LIN {X 0,Y 456.186,Z 1038.193,A -85,B 0,C 180,E1 14833.103,E2 14833.103} C_VEL
LIN {X 0,Y 454.706,Z 1048.98,A -85,B 0,C 180,E1 14838.466,E2 14838.466} C_VEL
LIN {X 0,Y 454.201,Z 1053.772,A -85,B 0,C 180,E1 14842.332,E2 14842.332} C_VEL
LIN {X 0,Y 454.081,Z 1056.363,A -85,B 0,C 180,E1 14848.088,E2 14848.088} C_VEL
LIN {X 0,Y 454.216,Z 1055.013,A -85,B 0,C 180,E1 14851.913,E2 14851.913} C_VEL
LIN {X 0,Y 454.611,Z 1049.888,A -85,B 0,C 180,E1 14856.701,E2 14856.701} C_VEL
LIN {X 0,Y 456.014,Z 1038.504,A -85,B 0,C 180,E1 14862.475,E2 14862.475} C_VEL
LIN {X 0,Y 459.25,Z 1020.736,A -85,B 0,C 180,E1 14868.27,E2 14868.27} C_VEL
LIN {X 0,Y 464.709,Z 997.367,A -85,B 0,C 180,E1 14873.669,E2 14873.669} C_VEL
LIN {X 0,Y 471.743,Z 970.349,A -85,B 0,C 180,E1 14878.315,E2 14878.315} C_VEL
LIN {X 0,Y 480.458,Z 937.273,A -85,B 0,C 180,E1 14882.614,E2 14882.614} C_VEL
LIN {X 0,Y 489.598,Z 900.461,A -85,B 0,C 180,E1 14886.199,E2 14886.199} C_VEL
LIN {X 0,Y 498.715,Z 857.606,A -85,B 0,C 180,E1 14889.265,E2 14889.265} C_VEL
LIN {X 0,Y 506.278,Z 812.153,A -85,B 0,C 180,E1 14891.552,E2 14891.552} C_VEL
LIN {X 0,Y 492.603,Z 777.017,A -85,B 0,C 180,E1 14894.833,E2 14894.833} C_VEL
LIN {X 0,Y 474.285,Z 742.388,A -85,B 0,C 180,E1 14898.475,E2 14898.475} C_VEL
LIN {X 0,Y 454.825,Z 713.013,A -85,B 0,C 180,E1 14902.271,E2 14902.271} C_VEL
LIN {X 0,Y 452.383,Z 707.31,A -85,B 0,C 180,E1 14902.914,E2 14902.914} C_VEL
LIN {X 0,Y 452.524,Z 707.31,A -85,B 0,C 180,E1 14909.843,E2 14909.843} C_VEL
LIN {X 0,Y 452.661,Z 707.31,A -85,B 0,C 180,E1 14916.31,E2 14916.31} C_VEL
LIN {X 0,Y 452.928,Z 707.31,A -85,B 0,C 180,E1 14922.472,E2 14922.472} C_VEL
LIN {X 0,Y 453.411,Z 707.31,A -85,B 0,C 180,E1 14928.428,E2 14928.428} C_VEL
LIN {X 0,Y 453.726,Z 707.31,A -85,B 0,C 180,E1 14934.246,E2 14934.246} C_VEL
LIN {X 0,Y 453.754,Z 707.31,A -85,B 0,C 180,E1 14941.91,E2 14941.91} C_VEL
LIN {X 0,Y 453.568,Z 707.31,A -85,B 0,C 180,E1 14947.677,E2 14947.677} C_VEL
LIN {X 0,Y 453.098,Z 707.31,A -85,B 0,C 180,E1 14954.087,E2 14954.087} C_VEL
LIN {X 0,Y 452.724,Z 707.31,A -85,B 0,C 180,E1 14960.404,E2 14960.404} C_VEL
LIN {X 0,Y 452.601,Z 707.31,A -85,B 0,C 180,E1 14965.798,E2 14965.798} C_VEL
LIN {X 0,Y 452.45,Z 707.31,A -85,B 0,C 180,E1 14972.4,E2 14972.4} C_VEL
LIN {X 0,Y 452.465,Z 708.154,A -85,B 0,C 180,E1 14974.776,E2 14974.776} C_VEL
LIN {X 0,Y 455.588,Z 713.626,A -85,B 0,C 180,E1 14975.457,E2 14975.457} C_VEL
LIN {X 0,Y 478.519,Z 749.077,A -85,B 0,C 180,E1 14979.815,E2 14979.815} C_VEL
LIN {X 0,Y 497.384,Z 784.719,A -85,B 0,C 180,E1 14983.272,E2 14983.272} C_VEL
LIN {X 0,Y 508.29,Z 812.813,A -85,B 0,C 180,E1 14985.653,E2 14985.653} C_VEL
LIN {X 0,Y 501.832,Z 855.362,A -85,B 0,C 180,E1 14987.392,E2 14987.392} C_VEL
LIN {X 0,Y 493.956,Z 895.887,A -85,B 0,C 180,E1 14989.745,E2 14989.745} C_VEL
LIN {X 0,Y 484.639,Z 936.283,A -85,B 0,C 180,E1 14992.968,E2 14992.968} C_VEL
LIN {X 0,Y 475.031,Z 974.706,A -85,B 0,C 180,E1 14997.157,E2 14997.157} C_VEL
LIN {X 0,Y 466.793,Z 1007.142,A -85,B 0,C 180,E1 15001.917,E2 15001.917} C_VEL
LIN {X 0,Y 460.332,Z 1035.051,A -85,B 0,C 180,E1 15007.471,E2 15007.471} C_VEL
LIN {X 0,Y 456.522,Z 1055.517,A -85,B 0,C 180,E1 15013.115,E2 15013.115} C_VEL
LIN {X 0,Y 454.835,Z 1068.915,A -85,B 0,C 180,E1 15018.468,E2 15018.468} C_VEL
LIN {X 0,Y 454.297,Z 1076.636,A -85,B 0,C 180,E1 15023.295,E2 15023.295} C_VEL
LIN {X 0,Y 454.154,Z 1080.28,A -85,B 0,C 180,E1 15028.087,E2 15028.087} C_VEL
LIN {X 0,Y 454.299,Z 1080.303,A -85,B 0,C 180,E1 15031.911,E2 15031.911} C_VEL
LIN {X 0,Y 454.27,Z 1075.566,A -85,B 0,C 180,E1 15037.667,E2 15037.667} C_VEL
LIN {X 0,Y 454.36,Z 1074.281,A -85,B 0,C 180,E1 15038.648,E2 15038.648} C_VEL
LIN {X 0,Y 450.707,Z 1070.833,A -85,B 0,C 180,E1 15040.771,E2 15040.771} C_VEL
LIN {X 0,Y 447.241,Z 1066.661,A -85,B 0,C 180,E1 15042.912,E2 15042.912} C_VEL
LIN {X 0,Y 449.59,Z 1051.412,A -85,B 0,C 180,E1 15048.62,E2 15048.62} C_VEL
LIN {X 0,Y 454.024,Z 1030.563,A -85,B 0,C 180,E1 15054.133,E2 15054.133} C_VEL
LIN {X 0,Y 460.882,Z 1004.236,A -85,B 0,C 180,E1 15059.28,E2 15059.28} C_VEL
LIN {X 0,Y 470.006,Z 971.713,A -85,B 0,C 180,E1 15064.022,E2 15064.022} C_VEL
LIN {X 0,Y 479.765,Z 935.941,A -85,B 0,C 180,E1 15067.932,E2 15067.932} C_VEL
LIN {X 0,Y 489.925,Z 894.816,A -85,B 0,C 180,E1 15071.239,E2 15071.239} C_VEL
LIN {X 0,Y 499.025,Z 850.387,A -85,B 0,C 180,E1 15073.79,E2 15073.79} C_VEL
LIN {X 0,Y 504.38,Z 814.102,A -85,B 0,C 180,E1 15075.308,E2 15075.308} C_VEL
LIN {X 0,Y 489.342,Z 779.423,A -85,B 0,C 180,E1 15078.711,E2 15078.711} C_VEL
LIN {X 0,Y 469.19,Z 744.618,A -85,B 0,C 180,E1 15082.806,E2 15082.806} C_VEL
LIN {X 0,Y 451.64,Z 719.415,A -85,B 0,C 180,E1 15086.659,E2 15086.659} C_VEL
LIN {X 0,Y 447.451,Z 713.438,A -85,B 0,C 180,E1 15087.687,E2 15087.687} C_VEL
LIN {X 0,Y 444.607,Z 708.574,A -85,B 0,C 180,E1 15088.439,E2 15088.439} C_VEL
LIN {X 0,Y 444.514,Z 707.31,A -85,B 0,C 180,E1 15088.637,E2 15088.637} C_VEL
LIN {X 0,Y 444.625,Z 707.31,A -85,B 0,C 180,E1 15093.704,E2 15093.704} C_VEL
LIN {X 0,Y 444.826,Z 707.31,A -85,B 0,C 180,E1 15100.086,E2 15100.086} C_VEL
LIN {X 0,Y 445.231,Z 707.31,A -85,B 0,C 180,E1 15106.22,E2 15106.22} C_VEL
LIN {X 0,Y 445.633,Z 707.31,A -85,B 0,C 180,E1 15112.186,E2 15112.186} C_VEL
LIN {X 0,Y 445.832,Z 707.31,A -85,B 0,C 180,E1 15118.056,E2 15118.056} C_VEL
LIN {X 0,Y 445.563,Z 707.31,A -85,B 0,C 180,E1 15123.904,E2 15123.904} C_VEL
LIN {X 0,Y 445.331,Z 707.31,A -85,B 0,C 180,E1 15129.8,E2 15129.8} C_VEL
LIN {X 0,Y 445.045,Z 707.31,A -85,B 0,C 180,E1 15135.811,E2 15135.811} C_VEL
LIN {X 0,Y 444.85,Z 707.31,A -85,B 0,C 180,E1 15142.01,E2 15142.01} C_VEL
LIN {X 0,Y 444.556,Z 707.31,A -85,B 0,C 180,E1 15149.224,E2 15149.224} C_VEL
LIN {X 0,Y 444.568,Z 707.532,A -85,B 0,C 180,E1 15149.854,E2 15149.854} C_VEL
LIN {X 0,Y 446.931,Z 712.981,A -85,B 0,C 180,E1 15150.524,E2 15150.524} C_VEL
LIN {X 0,Y 449.765,Z 716.523,A -85,B 0,C 180,E1 15151.214,E2 15151.214} C_VEL
LIN {X 0,Y 467.8,Z 742.864,A -85,B 0,C 180,E1 15155.295,E2 15155.295} C_VEL
LIN {X 0,Y 485.366,Z 773.688,A -85,B 0,C 180,E1 15159.154,E2 15159.154} C_VEL
LIN {X 0,Y 500.292,Z 808.905,A -85,B 0,C 180,E1 15162.897,E2 15162.897} C_VEL
LIN {X 0,Y 502.326,Z 818.223,A -85,B 0,C 180,E1 15163.698,E2 15163.698} C_VEL
LIN {X 0,Y 494.118,Z 861.819,A -85,B 0,C 180,E1 15165.968,E2 15165.968} C_VEL
LIN {X 0,Y 484.618,Z 902.54,A -85,B 0,C 180,E1 15168.955,E2 15168.955} C_VEL
LIN {X 0,Y 474.394,Z 940.654,A -85,B 0,C 180,E1 15172.785,E2 15172.785} C_VEL
LIN {X 0,Y 464.358,Z 975.438,A -85,B 0,C 180,E1 15177.533,E2 15177.533} C_VEL
LIN {X 0,Y 456.413,Z 1003.839,A -85,B 0,C 180,E1 15182.821,E2 15182.821} C_VEL
LIN {X 0,Y 450.631,Z 1027.018,A -85,B 0,C 180,E1 15188.808,E2 15188.808} C_VEL
LIN {X 0,Y 447.82,Z 1042.419,A -85,B 0,C 180,E1 15194.587,E2 15194.587} C_VEL
LIN {X 0,Y 446.526,Z 1051.875,A -85,B 0,C 180,E1 15200.231,E2 15200.231} C_VEL
LIN {X 0,Y 446.125,Z 1056.308,A -85,B 0,C 180,E1 15206.105,E2 15206.105} C_VEL
LIN {X 0,Y 446.415,Z 1056.23,A -85,B 0,C 180,E1 15210.001,E2 15210.001} C_VEL
LIN {X 0,Y 446.59,Z 1051.43,A -85,B 0,C 180,E1 15215.844,E2 15215.844} C_VEL
LIN {X 0,Y 447.898,Z 1041.018,A -85,B 0,C 180,E1 15221.713,E2 15221.713} C_VEL
LIN {X 0,Y 450.99,Z 1024.433,A -85,B 0,C 180,E1 15227.604,E2 15227.604} C_VEL
LIN {X 0,Y 456.366,Z 1001.802,A -85,B 0,C 180,E1 15233.224,E2 15233.224} C_VEL
LIN {X 0,Y 463.843,Z 973.876,A -85,B 0,C 180,E1 15238.306,E2 15238.306} C_VEL
LIN {X 0,Y 473.106,Z 940.161,A -85,B 0,C 180,E1 15242.856,E2 15242.856} C_VEL
LIN {X 0,Y 483.21,Z 900.916,A -85,B 0,C 180,E1 15246.756,E2 15246.756} C_VEL
LIN {X 0,Y 492.663,Z 857.898,A -85,B 0,C 180,E1 15249.862,E2 15249.862} C_VEL
LIN {X 0,Y 500.04,Z 814.852,A -85,B 0,C 180,E1 15252.07,E2 15252.07} C_VEL
LIN {X 0,Y 486.137,Z 778.648,A -85,B 0,C 180,E1 15255.57,E2 15255.57} C_VEL
LIN {X 0,Y 467.182,Z 743.055,A -85,B 0,C 180,E1 15259.499,E2 15259.499} C_VEL
LIN {X 0,Y 447.132,Z 713.195,A -85,B 0,C 180,E1 15263.624,E2 15263.624} C_VEL
LIN {X 0,Y 444.506,Z 708.118,A -85,B 0,C 180,E1 15264.25,E2 15264.25} C_VEL
LIN {X 0,Y 444.531,Z 707.31,A -85,B 0,C 180,E1 15269.243,E2 15269.243} C_VEL
LIN {X 0,Y 444.743,Z 707.31,A -85,B 0,C 180,E1 15275.862,E2 15275.862} C_VEL
LIN {X 0,Y 445.023,Z 707.31,A -85,B 0,C 180,E1 15282.454,E2 15282.454} C_VEL
LIN {X 0,Y 445.484,Z 707.31,A -85,B 0,C 180,E1 15288.22,E2 15288.22} C_VEL
LIN {X 0,Y 445.805,Z 707.31,A -85,B 0,C 180,E1 15294.143,E2 15294.143} C_VEL
LIN {X 0,Y 445.841,Z 707.31,A -85,B 0,C 180,E1 15301.944,E2 15301.944} C_VEL
LIN {X 0,Y 445.647,Z 707.31,A -85,B 0,C 180,E1 15307.814,E2 15307.814} C_VEL
LIN {X 0,Y 445.244,Z 707.31,A -85,B 0,C 180,E1 15313.779,E2 15313.779} C_VEL
LIN {X 0,Y 444.836,Z 707.31,A -85,B 0,C 180,E1 15319.913,E2 15319.913} C_VEL
LIN {X 0,Y 444.632,Z 707.31,A -85,B 0,C 180,E1 15326.295,E2 15326.295} C_VEL
LIN {X 0,Y 444.507,Z 707.31,A -85,B 0,C 180,E1 15333.284,E2 15333.284} C_VEL
LIN {X 0,Y 446.827,Z 712.942,A -85,B 0,C 180,E1 15333.896,E2 15333.896} C_VEL
LIN {X 0,Y 449.926,Z 717.277,A -85,B 0,C 180,E1 15334.572,E2 15334.572} C_VEL
LIN {X 0,Y 468.229,Z 744.574,A -85,B 0,C 180,E1 15338.234,E2 15338.234} C_VEL
LIN {X 0,Y 488.407,Z 781.004,A -85,B 0,C 180,E1 15342.056,E2 15342.056} C_VEL
LIN {X 0,Y 502.202,Z 814.372,A -85,B 0,C 180,E1 15345.071,E2 15345.071} C_VEL
LIN {X 0,Y 495.094,Z 859.617,A -85,B 0,C 180,E1 15346.999,E2 15346.999} C_VEL
LIN {X 0,Y 487.037,Z 898.739,A -85,B 0,C 180,E1 15349.362,E2 15349.362} C_VEL
LIN {X 0,Y 477.602,Z 938.053,A -85,B 0,C 180,E1 15352.589,E2 15352.589} C_VEL
LIN {X 0,Y 468.18,Z 974.379,A -85,B 0,C 180,E1 15356.615,E2 15356.615} C_VEL
LIN {X 0,Y 459.534,Z 1006.996,A -85,B 0,C 180,E1 15361.463,E2 15361.463} C_VEL
LIN {X 0,Y 453.069,Z 1033.593,A -85,B 0,C 180,E1 15366.801,E2 15366.801} C_VEL
LIN {X 0,Y 448.77,Z 1055.256,A -85,B 0,C 180,E1 15372.813,E2 15372.813} C_VEL
LIN {X 0,Y 446.971,Z 1068.675,A -85,B 0,C 180,E1 15378.262,E2 15378.262} C_VEL
LIN {X 0,Y 446.409,Z 1076.408,A -85,B 0,C 180,E1 15383.176,E2 15383.176} C_VEL
LIN {X 0,Y 446.252,Z 1080.066,A -85,B 0,C 180,E1 15388.053,E2 15388.053} C_VEL
LIN {X 0,Y 446.395,Z 1080.094,A -85,B 0,C 180,E1 15391.945,E2 15391.945} C_VEL
LIN {X 0,Y 446.375,Z 1075.37,A -85,B 0,C 180,E1 15397.804,E2 15397.804} C_VEL
LIN {X 0,Y 447.241,Z 1066.661,A -85,B 0,C 180,E1 15402.912,E2 15402.912} C_VEL
LIN {X 0,Y 443.939,Z 1061.938,A -85,B 0,C 180,E1 15405.041,E2 15405.041} C_VEL
LIN {X 0,Y 440.957,Z 1056.558,A -85,B 0,C 180,E1 15407.179,E2 15407.179} C_VEL
LIN {X 0,Y 445.138,Z 1036.482,A -85,B 0,C 180,E1 15413.104,E2 15413.104} C_VEL
LIN {X 0,Y 451.671,Z 1011.412,A -85,B 0,C 180,E1 15418.479,E2 15418.479} C_VEL
LIN {X 0,Y 460.159,Z 982.234,A -85,B 0,C 180,E1 15423.166,E2 15423.166} C_VEL
LIN {X 0,Y 470.066,Z 947.885,A -85,B 0,C 180,E1 15427.334,E2 15427.334} C_VEL
LIN {X 0,Y 480.939,Z 906.832,A -85,B 0,C 180,E1 15431.004,E2 15431.004} C_VEL
LIN {X 0,Y 490.884,Z 863.211,A -85,B 0,C 180,E1 15433.786,E2 15433.786} C_VEL
LIN {X 0,Y 498.525,Z 817.345,A -85,B 0,C 180,E1 15435.837,E2 15435.837} C_VEL
LIN {X 0,Y 483.899,Z 783.034,A -85,B 0,C 180,E1 15439.334,E2 15439.334} C_VEL
LIN {X 0,Y 465.253,Z 750.222,A -85,B 0,C 180,E1 15443.315,E2 15443.315} C_VEL
LIN {X 0,Y 444.926,Z 720.523,A -85,B 0,C 180,E1 15448.004,E2 15448.004} C_VEL
LIN {X 0,Y 439.645,Z 713.508,A -85,B 0,C 180,E1 15449.383,E2 15449.383} C_VEL
LIN {X 0,Y 436.726,Z 708.582,A -85,B 0,C 180,E1 15450.22,E2 15450.22} C_VEL
LIN {X 0,Y 436.609,Z 707.31,A -85,B 0,C 180,E1 15450.436,E2 15450.436} C_VEL
LIN {X 0,Y 436.827,Z 707.31,A -85,B 0,C 180,E1 15457.571,E2 15457.571} C_VEL
LIN {X 0,Y 437.121,Z 707.31,A -85,B 0,C 180,E1 15463.902,E2 15463.902} C_VEL
LIN {X 0,Y 437.639,Z 707.31,A -85,B 0,C 180,E1 15470.034,E2 15470.034} C_VEL
LIN {X 0,Y 437.672,Z 707.31,A -85,B 0,C 180,E1 15476.033,E2 15476.033} C_VEL
LIN {X 0,Y 437.618,Z 707.31,A -85,B 0,C 180,E1 15481.988,E2 15481.988} C_VEL
LIN {X 0,Y 437.455,Z 707.31,A -85,B 0,C 180,E1 15487.968,E2 15487.968} C_VEL
LIN {X 0,Y 437.277,Z 707.31,A -85,B 0,C 180,E1 15494.043,E2 15494.043} C_VEL
LIN {X 0,Y 436.933,Z 707.31,A -85,B 0,C 180,E1 15500.542,E2 15500.542} C_VEL
LIN {X 0,Y 436.643,Z 707.31,A -85,B 0,C 180,E1 15507.476,E2 15507.476} C_VEL
LIN {X 0,Y 436.677,Z 708.191,A -85,B 0,C 180,E1 15508.089,E2 15508.089} C_VEL
LIN {X 0,Y 439.613,Z 713.446,A -85,B 0,C 180,E1 15508.942,E2 15508.942} C_VEL
LIN {X 0,Y 442.067,Z 716.673,A -85,B 0,C 180,E1 15509.593,E2 15509.593} C_VEL
LIN {X 0,Y 459.278,Z 741.265,A -85,B 0,C 180,E1 15513.764,E2 15513.764} C_VEL
LIN {X 0,Y 477.735,Z 772.896,A -85,B 0,C 180,E1 15518.011,E2 15518.011} C_VEL
LIN {X 0,Y 492.517,Z 807.026,A -85,B 0,C 180,E1 15521.828,E2 15521.828} C_VEL
LIN {X 0,Y 496.591,Z 819.004,A -85,B 0,C 180,E1 15523.066,E2 15523.066} C_VEL
LIN {X 0,Y 488.32,Z 861.92,A -85,B 0,C 180,E1 15525.323,E2 15525.323} C_VEL
LIN {X 0,Y 478.532,Z 902.526,A -85,B 0,C 180,E1 15528.317,E2 15528.317} C_VEL
LIN {X 0,Y 467.903,Z 940.684,A -85,B 0,C 180,E1 15532.179,E2 15532.179} C_VEL
LIN {X 0,Y 457.703,Z 974.903,A -85,B 0,C 180,E1 15536.888,E2 15536.888} C_VEL
LIN {X 0,Y 449.079,Z 1004.023,A -85,B 0,C 180,E1 15542.356,E2 15542.356} C_VEL
LIN {X 0,Y 443.037,Z 1027.164,A -85,B 0,C 180,E1 15548.427,E2 15548.427} C_VEL
LIN {X 0,Y 440.099,Z 1041.922,A -85,B 0,C 180,E1 15554.011,E2 15554.011} C_VEL
LIN {X 0,Y 438.821,Z 1050.866,A -85,B 0,C 180,E1 15559.052,E2 15559.052} C_VEL
LIN {X 0,Y 438.263,Z 1055.639,A -85,B 0,C 180,E1 15564.047,E2 15564.047} C_VEL
LIN {X 0,Y 438.533,Z 1056.446,A -85,B 0,C 180,E1 15570.001,E2 15570.001} C_VEL
LIN {X 0,Y 438.724,Z 1051.669,A -85,B 0,C 180,E1 15575.949,E2 15575.949} C_VEL
LIN {X 0,Y 439.819,Z 1043.03,A -85,B 0,C 180,E1 15581.15,E2 15581.15} C_VEL
LIN {X 0,Y 443.037,Z 1026.246,A -85,B 0,C 180,E1 15587.471,E2 15587.471} C_VEL
LIN {X 0,Y 448.683,Z 1003.307,A -85,B 0,C 180,E1 15593.382,E2 15593.382} C_VEL
LIN {X 0,Y 456.726,Z 974.533,A -85,B 0,C 180,E1 15598.736,E2 15598.736} C_VEL
LIN {X 0,Y 466.408,Z 940.559,A -85,B 0,C 180,E1 15603.389,E2 15603.389} C_VEL
LIN {X 0,Y 476.835,Z 901.541,A -85,B 0,C 180,E1 15607.312,E2 15607.312} C_VEL
LIN {X 0,Y 486.484,Z 859.193,A -85,B 0,C 180,E1 15610.413,E2 15610.413} C_VEL
LIN {X 0,Y 493.876,Z 817.882,A -85,B 0,C 180,E1 15612.569,E2 15612.569} C_VEL
LIN {X 0,Y 480.27,Z 781.639,A -85,B 0,C 180,E1 15616.201,E2 15616.201} C_VEL
LIN {X 0,Y 462.388,Z 747.702,A -85,B 0,C 180,E1 15620.099,E2 15620.099} C_VEL
LIN {X 0,Y 443.563,Z 719.344,A -85,B 0,C 180,E1 15624.113,E2 15624.113} C_VEL
LIN {X 0,Y 439,Z 713.014,A -85,B 0,C 180,E1 15625.17,E2 15625.17} C_VEL
LIN {X 0,Y 436.537,Z 707.31,A -85,B 0,C 180,E1 15626.008,E2 15626.008} C_VEL
LIN {X 0,Y 436.697,Z 707.31,A -85,B 0,C 180,E1 15633.181,E2 15633.181} C_VEL
LIN {X 0,Y 436.905,Z 707.31,A -85,B 0,C 180,E1 15639.702,E2 15639.702} C_VEL
LIN {X 0,Y 437.383,Z 707.31,A -85,B 0,C 180,E1 15645.961,E2 15645.961} C_VEL
LIN {X 0,Y 437.749,Z 707.31,A -85,B 0,C 180,E1 15652.037,E2 15652.037} C_VEL
LIN {X 0,Y 437.643,Z 707.31,A -85,B 0,C 180,E1 15658.012,E2 15658.012} C_VEL
LIN {X 0,Y 437.67,Z 707.31,A -85,B 0,C 180,E1 15663.967,E2 15663.967} C_VEL
LIN {X 0,Y 437.653,Z 707.31,A -85,B 0,C 180,E1 15669.966,E2 15669.966} C_VEL
LIN {X 0,Y 437.133,Z 707.31,A -85,B 0,C 180,E1 15676.097,E2 15676.097} C_VEL
LIN {X 0,Y 436.839,Z 707.31,A -85,B 0,C 180,E1 15682.428,E2 15682.428} C_VEL
LIN {X 0,Y 436.644,Z 707.31,A -85,B 0,C 180,E1 15689.066,E2 15689.066} C_VEL
LIN {X 0,Y 436.634,Z 707.318,A -85,B 0,C 180,E1 15691.773,E2 15691.773} C_VEL
LIN {X 0,Y 438.701,Z 712.684,A -85,B 0,C 180,E1 15692.344,E2 15692.344} C_VEL
LIN {X 0,Y 441.686,Z 716.541,A -85,B 0,C 180,E1 15693.035,E2 15693.035} C_VEL
LIN {X 0,Y 461.26,Z 745.525,A -85,B 0,C 180,E1 15697.188,E2 15697.188} C_VEL
LIN {X 0,Y 480.502,Z 779.804,A -85,B 0,C 180,E1 15701.003,E2 15701.003} C_VEL
LIN {X 0,Y 495.946,Z 816.725,A -85,B 0,C 180,E1 15704.492,E2 15704.492} C_VEL
LIN {X 0,Y 488.248,Z 864.434,A -85,B 0,C 180,E1 15706.629,E2 15706.629} C_VEL
LIN {X 0,Y 478.889,Z 907.156,A -85,B 0,C 180,E1 15709.373,E2 15709.373} C_VEL
LIN {X 0,Y 468.621,Z 947.439,A -85,B 0,C 180,E1 15712.965,E2 15712.965} C_VEL
LIN {X 0,Y 458.67,Z 983.652,A -85,B 0,C 180,E1 15717.358,E2 15717.358} C_VEL
LIN {X 0,Y 450.507,Z 1013.662,A -85,B 0,C 180,E1 15722.251,E2 15722.251} C_VEL
LIN {X 0,Y 444.354,Z 1038.417,A -85,B 0,C 180,E1 15727.66,E2 15727.66} C_VEL
LIN {X 0,Y 440.773,Z 1056.435,A -85,B 0,C 180,E1 15733.007,E2 15733.007} C_VEL
LIN {X 0,Y 438.995,Z 1069.765,A -85,B 0,C 180,E1 15738.729,E2 15738.729} C_VEL
LIN {X 0,Y 438.483,Z 1077.216,A -85,B 0,C 180,E1 15744.048,E2 15744.048} C_VEL
LIN {X 0,Y 438.512,Z 1080.206,A -85,B 0,C 180,E1 15749.999,E2 15749.999} C_VEL
LIN {X 0,Y 438.47,Z 1077.374,A -85,B 0,C 180,E1 15755.95,E2 15755.95} C_VEL
LIN {X 0,Y 438.943,Z 1070.23,A -85,B 0,C 180,E1 15761.235,E2 15761.235} C_VEL
LIN {X 0,Y 440.957,Z 1056.558,A -85,B 0,C 180,E1 15767.179,E2 15767.179} C_VEL
LIN {X 0,Y 438.256,Z 1050.682,A -85,B 0,C 180,E1 15769.303,E2 15769.303} C_VEL
LIN {X 0,Y 435.819,Z 1044.111,A -85,B 0,C 180,E1 15771.419,E2 15771.419} C_VEL
LIN {X 0,Y 441.902,Z 1020.734,A -85,B 0,C 180,E1 15777.102,E2 15777.102} C_VEL
LIN {X 0,Y 449.922,Z 993.481,A -85,B 0,C 180,E1 15782.037,E2 15782.037} C_VEL
LIN {X 0,Y 460.181,Z 959.48,A -85,B 0,C 180,E1 15786.645,E2 15786.645} C_VEL
LIN {X 0,Y 471.284,Z 920.476,A -85,B 0,C 180,E1 15790.54,E2 15790.54} C_VEL
LIN {X 0,Y 482.028,Z 877.609,A -85,B 0,C 180,E1 15793.621,E2 15793.621} C_VEL
LIN {X 0,Y 491.151,Z 832.43,A -85,B 0,C 180,E1 15795.87,E2 15795.87} C_VEL
LIN {X 0,Y 492.497,Z 819.986,A -85,B 0,C 180,E1 15796.421,E2 15796.421} C_VEL
LIN {X 0,Y 478.235,Z 786.157,A -85,B 0,C 180,E1 15800.004,E2 15800.004} C_VEL
LIN {X 0,Y 460.352,Z 754.369,A -85,B 0,C 180,E1 15804.033,E2 15804.033} C_VEL
LIN {X 0,Y 441.618,Z 726.789,A -85,B 0,C 180,E1 15808.523,E2 15808.523} C_VEL
LIN {X 0,Y 432.417,Z 713.971,A -85,B 0,C 180,E1 15811.08,E2 15811.08} C_VEL
LIN {X 0,Y 428.934,Z 709.282,A -85,B 0,C 180,E1 15812.131,E2 15812.131} C_VEL
LIN {X 0,Y 428.702,Z 707.31,A -85,B 0,C 180,E1 15812.414,E2 15812.414} C_VEL
LIN {X 0,Y 428.939,Z 707.31,A -85,B 0,C 180,E1 15819.316,E2 15819.316} C_VEL
LIN {X 0,Y 429.337,Z 707.31,A -85,B 0,C 180,E1 15825.7,E2 15825.7} C_VEL
LIN {X 0,Y 429.79,Z 707.31,A -85,B 0,C 180,E1 15831.896,E2 15831.896} C_VEL
LIN {X 0,Y 430.011,Z 707.31,A -85,B 0,C 180,E1 15837.984,E2 15837.984} C_VEL
LIN {X 0,Y 429.74,Z 707.31,A -85,B 0,C 180,E1 15844.048,E2 15844.048} C_VEL
LIN {X 0,Y 429.498,Z 707.31,A -85,B 0,C 180,E1 15850.165,E2 15850.165} C_VEL
LIN {X 0,Y 429.163,Z 707.31,A -85,B 0,C 180,E1 15856.412,E2 15856.412} C_VEL
LIN {X 0,Y 428.901,Z 707.31,A -85,B 0,C 180,E1 15863.275,E2 15863.275} C_VEL
LIN {X 0,Y 428.772,Z 707.433,A -85,B 0,C 180,E1 15866.094,E2 15866.094} C_VEL
LIN {X 0,Y 430.827,Z 712.624,A -85,B 0,C 180,E1 15866.808,E2 15866.808} C_VEL
LIN {X 0,Y 434.1,Z 716.27,A -85,B 0,C 180,E1 15867.744,E2 15867.744} C_VEL
LIN {X 0,Y 451.862,Z 741.347,A -85,B 0,C 180,E1 15872.382,E2 15872.382} C_VEL
LIN {X 0,Y 470.793,Z 773.323,A -85,B 0,C 180,E1 15876.968,E2 15876.968} C_VEL
LIN {X 0,Y 485.624,Z 807.281,A -85,B 0,C 180,E1 15880.947,E2 15880.947} C_VEL
LIN {X 0,Y 490.548,Z 822.804,A -85,B 0,C 180,E1 15882.573,E2 15882.573} C_VEL
LIN {X 0,Y 482.12,Z 863.975,A -85,B 0,C 180,E1 15884.79,E2 15884.79} C_VEL
LIN {X 0,Y 472.154,Z 903.798,A -85,B 0,C 180,E1 15887.78,E2 15887.78} C_VEL
LIN {X 0,Y 461.125,Z 941.939,A -85,B 0,C 180,E1 15891.703,E2 15891.703} C_VEL
LIN {X 0,Y 450.846,Z 974.977,A -85,B 0,C 180,E1 15896.318,E2 15896.318} C_VEL
LIN {X 0,Y 441.817,Z 1004.137,A -85,B 0,C 180,E1 15901.862,E2 15901.862} C_VEL
LIN {X 0,Y 435.485,Z 1027.311,A -85,B 0,C 180,E1 15908.034,E2 15908.034} C_VEL
LIN {X 0,Y 432.126,Z 1043.636,A -85,B 0,C 180,E1 15914.427,E2 15914.427} C_VEL
LIN {X 0,Y 430.784,Z 1052.48,A -85,B 0,C 180,E1 15920.073,E2 15920.073} C_VEL
LIN {X 0,Y 430.342,Z 1056.723,A -85,B 0,C 180,E1 15925.962,E2 15925.962} C_VEL
LIN {X 0,Y 430.632,Z 1056.661,A -85,B 0,C 180,E1 15930.001,E2 15930.001} C_VEL
LIN {X 0,Y 430.843,Z 1051.908,A -85,B 0,C 180,E1 15936.058,E2 15936.058} C_VEL
LIN {X 0,Y 431.986,Z 1043.515,A -85,B 0,C 180,E1 15941.254,E2 15941.254} C_VEL
LIN {X 0,Y 435.344,Z 1026.723,A -85,B 0,C 180,E1 15947.734,E2 15947.734} C_VEL
LIN {X 0,Y 441.287,Z 1003.631,A -85,B 0,C 180,E1 15953.798,E2 15953.798} C_VEL
LIN {X 0,Y 449.747,Z 974.698,A -85,B 0,C 180,E1 15959.259,E2 15959.259} C_VEL
LIN {X 0,Y 459.731,Z 940.957,A -85,B 0,C 180,E1 15963.94,E2 15963.94} C_VEL
LIN {X 0,Y 470.543,Z 901.992,A -85,B 0,C 180,E1 15967.898,E2 15967.898} C_VEL
LIN {X 0,Y 480.557,Z 859.406,A -85,B 0,C 180,E1 15971.043,E2 15971.043} C_VEL
LIN {X 0,Y 487.619,Z 820.313,A -85,B 0,C 180,E1 15973.135,E2 15973.135} C_VEL
LIN {X 0,Y 474.166,Z 784.229,A -85,B 0,C 180,E1 15976.888,E2 15976.888} C_VEL
LIN {X 0,Y 456.53,Z 750.238,A -85,B 0,C 180,E1 15980.954,E2 15980.954} C_VEL
LIN {X 0,Y 436.596,Z 720.251,A -85,B 0,C 180,E1 15985.435,E2 15985.435} C_VEL
LIN {X 0,Y 431.409,Z 713.289,A -85,B 0,C 180,E1 15986.714,E2 15986.714} C_VEL
LIN {X 0,Y 428.731,Z 708.643,A -85,B 0,C 180,E1 15987.438,E2 15987.438} C_VEL
LIN {X 0,Y 428.644,Z 707.31,A -85,B 0,C 180,E1 15987.701,E2 15987.701} C_VEL
LIN {X 0,Y 428.835,Z 707.31,A -85,B 0,C 180,E1 15994.906,E2 15994.906} C_VEL
LIN {X 0,Y 429.087,Z 707.31,A -85,B 0,C 180,E1 16001.463,E2 16001.463} C_VEL
LIN {X 0,Y 429.601,Z 707.31,A -85,B 0,C 180,E1 16007.777,E2 16007.777} C_VEL
LIN {X 0,Y 429.96,Z 707.31,A -85,B 0,C 180,E1 16013.927,E2 16013.927} C_VEL
LIN {X 0,Y 430.02,Z 707.31,A -85,B 0,C 180,E1 16022.016,E2 16022.016} C_VEL
LIN {X 0,Y 429.72,Z 707.31,A -85,B 0,C 180,E1 16029.095,E2 16029.095} C_VEL
LIN {X 0,Y 429.35,Z 707.31,A -85,B 0,C 180,E1 16034.3,E2 16034.3} C_VEL
LIN {X 0,Y 428.95,Z 707.31,A -85,B 0,C 180,E1 16040.684,E2 16040.684} C_VEL
LIN {X 0,Y 428.7,Z 707.31,A -85,B 0,C 180,E1 16047.904,E2 16047.904} C_VEL
LIN {X 0,Y 428.744,Z 708.006,A -85,B 0,C 180,E1 16050.127,E2 16050.127} C_VEL
LIN {X 0,Y 431.498,Z 713.334,A -85,B 0,C 180,E1 16050.889,E2 16050.889} C_VEL
LIN {X 0,Y 434.188,Z 717.076,A -85,B 0,C 180,E1 16051.565,E2 16051.565} C_VEL
LIN {X 0,Y 452.302,Z 743.403,A -85,B 0,C 180,E1 16055.673,E2 16055.673} C_VEL
LIN {X 0,Y 471.39,Z 776.156,A -85,B 0,C 180,E1 16059.636,E2 16059.636} C_VEL
LIN {X 0,Y 486.953,Z 811.593,A -85,B 0,C 180,E1 16063.202,E2 16063.202} C_VEL
LIN {X 0,Y 489.952,Z 820.648,A -85,B 0,C 180,E1 16064.026,E2 16064.026} C_VEL
LIN {X 0,Y 482.011,Z 865.908,A -85,B 0,C 180,E1 16066.082,E2 16066.082} C_VEL
LIN {X 0,Y 472.596,Z 907.562,A -85,B 0,C 180,E1 16068.796,E2 16068.796} C_VEL
LIN {X 0,Y 461.832,Z 948.242,A -85,B 0,C 180,E1 16072.475,E2 16072.475} C_VEL
LIN {X 0,Y 451.186,Z 985.461,A -85,B 0,C 180,E1 16077.098,E2 16077.098} C_VEL
LIN {X 0,Y 442.363,Z 1016.819,A -85,B 0,C 180,E1 16082.418,E2 16082.418} C_VEL
LIN {X 0,Y 436.084,Z 1041.278,A -85,B 0,C 180,E1 16088.063,E2 16088.063} C_VEL
LIN {X 0,Y 432.294,Z 1060.809,A -85,B 0,C 180,E1 16094.439,E2 16094.439} C_VEL
LIN {X 0,Y 430.909,Z 1071.888,A -85,B 0,C 180,E1 16099.936,E2 16099.936} C_VEL
LIN {X 0,Y 430.583,Z 1076.992,A -85,B 0,C 180,E1 16103.938,E2 16103.938} C_VEL
LIN {X 0,Y 430.613,Z 1079.992,A -85,B 0,C 180,E1 16109.999,E2 16109.999} C_VEL
LIN {X 0,Y 430.566,Z 1077.174,A -85,B 0,C 180,E1 16116.06,E2 16116.06} C_VEL
LIN {X 0,Y 431.022,Z 1070.545,A -85,B 0,C 180,E1 16121.149,E2 16121.149} C_VEL
LIN {X 0,Y 433.119,Z 1056.896,A -85,B 0,C 180,E1 16127.3,E2 16127.3} C_VEL
LIN {X 0,Y 435.819,Z 1044.111,A -85,B 0,C 180,E1 16131.419,E2 16131.419} C_VEL
LIN {X 0,Y 433.636,Z 1037.147,A -85,B 0,C 180,E1 16133.525,E2 16133.525} C_VEL
LIN {X 0,Y 432.023,Z 1029.493,A -85,B 0,C 180,E1 16135.603,E2 16135.603} C_VEL
LIN {X 0,Y 439.796,Z 1003.772,A -85,B 0,C 180,E1 16140.849,E2 16140.849} C_VEL
LIN {X 0,Y 449.778,Z 972.088,A -85,B 0,C 180,E1 16145.678,E2 16145.678} C_VEL
LIN {X 0,Y 461.124,Z 935.021,A -85,B 0,C 180,E1 16149.853,E2 16149.853} C_VEL
LIN {X 0,Y 472.606,Z 892.853,A -85,B 0,C 180,E1 16153.3,E2 16153.3} C_VEL
LIN {X 0,Y 482.54,Z 848.694,A -85,B 0,C 180,E1 16155.839,E2 16155.839} C_VEL
LIN {X 0,Y 486.762,Z 823.646,A -85,B 0,C 180,E1 16156.929,E2 16156.929} C_VEL
LIN {X 0,Y 473.137,Z 790.544,A -85,B 0,C 180,E1 16160.557,E2 16160.557} C_VEL
LIN {X 0,Y 455.558,Z 758.244,A -85,B 0,C 180,E1 16164.77,E2 16164.77} C_VEL
LIN {X 0,Y 437.911,Z 732.421,A -85,B 0,C 180,E1 16169.168,E2 16169.168} C_VEL
LIN {X 0,Y 429.107,Z 720.377,A -85,B 0,C 180,E1 16171.689,E2 16171.689} C_VEL
LIN {X 0,Y 424.554,Z 714.045,A -85,B 0,C 180,E1 16173.13,E2 16173.13} C_VEL
LIN {X 0,Y 421.086,Z 709.323,A -85,B 0,C 180,E1 16174.297,E2 16174.297} C_VEL
LIN {X 0,Y 420.859,Z 707.31,A -85,B 0,C 180,E1 16174.547,E2 16174.547} C_VEL
LIN {X 0,Y 421.087,Z 707.31,A -85,B 0,C 180,E1 16181.106,E2 16181.106} C_VEL
LIN {X 0,Y 421.562,Z 707.31,A -85,B 0,C 180,E1 16187.548,E2 16187.548} C_VEL
LIN {X 0,Y 421.878,Z 707.31,A -85,B 0,C 180,E1 16193.818,E2 16193.818} C_VEL
LIN {X 0,Y 422.127,Z 707.31,A -85,B 0,C 180,E1 16200.004,E2 16200.004} C_VEL
LIN {X 0,Y 421.756,Z 707.31,A -85,B 0,C 180,E1 16206.192,E2 16206.192} C_VEL
LIN {X 0,Y 421.483,Z 707.31,A -85,B 0,C 180,E1 16212.462,E2 16212.462} C_VEL
LIN {X 0,Y 421.141,Z 707.31,A -85,B 0,C 180,E1 16218.9,E2 16218.9} C_VEL
LIN {X 0,Y 420.94,Z 707.498,A -85,B 0,C 180,E1 16223.921,E2 16223.921} C_VEL
LIN {X 0,Y 422.918,Z 712.571,A -85,B 0,C 180,E1 16224.691,E2 16224.691} C_VEL
LIN {X 0,Y 426.299,Z 716.076,A -85,B 0,C 180,E1 16225.754,E2 16225.754} C_VEL
LIN {X 0,Y 441.848,Z 737.915,A -85,B 0,C 180,E1 16230.222,E2 16230.222} C_VEL
LIN {X 0,Y 459.184,Z 765.382,A -85,B 0,C 180,E1 16234.662,E2 16234.662} C_VEL
LIN {X 0,Y 474.58,Z 796.828,A -85,B 0,C 180,E1 16238.771,E2 16238.771} C_VEL
LIN {X 0,Y 484.467,Z 824.476,A -85,B 0,C 180,E1 16241.914,E2 16241.914} C_VEL
LIN {X 0,Y 475.82,Z 866.647,A -85,B 0,C 180,E1 16244.283,E2 16244.283} C_VEL
LIN {X 0,Y 465.802,Z 905.06,A -85,B 0,C 180,E1 16247.226,E2 16247.226} C_VEL
LIN {X 0,Y 454.862,Z 941.601,A -85,B 0,C 180,E1 16251.018,E2 16251.018} C_VEL
LIN {X 0,Y 444.024,Z 975.053,A -85,B 0,C 180,E1 16255.729,E2 16255.729} C_VEL
LIN {X 0,Y 434.574,Z 1004.25,A -85,B 0,C 180,E1 16261.35,E2 16261.35} C_VEL
LIN {X 0,Y 427.942,Z 1027.458,A -85,B 0,C 180,E1 16267.626,E2 16267.626} C_VEL
LIN {X 0,Y 424.349,Z 1043.858,A -85,B 0,C 180,E1 16274.163,E2 16274.163} C_VEL
LIN {X 0,Y 422.944,Z 1052.43,A -85,B 0,C 180,E1 16279.681,E2 16279.681} C_VEL
LIN {X 0,Y 422.444,Z 1056.93,A -85,B 0,C 180,E1 16285.887,E2 16285.887} C_VEL
LIN {X 0,Y 422.761,Z 1056.875,A -85,B 0,C 180,E1 16290.001,E2 16290.001} C_VEL
LIN {X 0,Y 422.963,Z 1052.147,A -85,B 0,C 180,E1 16296.171,E2 16296.171} C_VEL
LIN {X 0,Y 424.214,Z 1043.459,A -85,B 0,C 180,E1 16301.612,E2 16301.612} C_VEL
LIN {X 0,Y 427.712,Z 1027.015,A -85,B 0,C 180,E1 16308.061,E2 16308.061} C_VEL
LIN {X 0,Y 433.941,Z 1003.953,A -85,B 0,C 180,E1 16314.227,E2 16314.227} C_VEL
LIN {X 0,Y 442.73,Z 975.116,A -85,B 0,C 180,E1 16319.757,E2 16319.757} C_VEL
LIN {X 0,Y 453.416,Z 940.316,A -85,B 0,C 180,E1 16324.624,E2 16324.624} C_VEL
LIN {X 0,Y 464.216,Z 902.662,A -85,B 0,C 180,E1 16328.484,E2 16328.484} C_VEL
LIN {X 0,Y 474.711,Z 859.487,A -85,B 0,C 180,E1 16331.697,E2 16331.697} C_VEL
LIN {X 0,Y 481.588,Z 823.671,A -85,B 0,C 180,E1 16333.632,E2 16333.632} C_VEL
LIN {X 0,Y 468.785,Z 788.331,A -85,B 0,C 180,E1 16337.415,E2 16337.415} C_VEL
LIN {X 0,Y 451.969,Z 755.328,A -85,B 0,C 180,E1 16341.505,E2 16341.505} C_VEL
LIN {X 0,Y 433.36,Z 726.69,A -85,B 0,C 180,E1 16345.899,E2 16345.899} C_VEL
LIN {X 0,Y 423.883,Z 713.631,A -85,B 0,C 180,E1 16348.369,E2 16348.369} C_VEL
LIN {X 0,Y 420.872,Z 708.977,A -85,B 0,C 180,E1 16349.234,E2 16349.234} C_VEL
LIN {X 0,Y 420.712,Z 707.31,A -85,B 0,C 180,E1 16349.432,E2 16349.432} C_VEL
LIN {X 0,Y 420.973,Z 707.31,A -85,B 0,C 180,E1 16356.67,E2 16356.67} C_VEL
LIN {X 0,Y 421.298,Z 707.31,A -85,B 0,C 180,E1 16363.273,E2 16363.273} C_VEL
LIN {X 0,Y 421.825,Z 707.31,A -85,B 0,C 180,E1 16369.648,E2 16369.648} C_VEL
LIN {X 0,Y 421.976,Z 707.31,A -85,B 0,C 180,E1 16375.878,E2 16375.878} C_VEL
LIN {X 0,Y 422.119,Z 707.31,A -85,B 0,C 180,E1 16382.054,E2 16382.054} C_VEL
LIN {X 0,Y 421.891,Z 707.31,A -85,B 0,C 180,E1 16388.257,E2 16388.257} C_VEL
LIN {X 0,Y 421.419,Z 707.31,A -85,B 0,C 180,E1 16394.575,E2 16394.575} C_VEL
LIN {X 0,Y 420.989,Z 707.31,A -85,B 0,C 180,E1 16401.094,E2 16401.094} C_VEL
LIN {X 0,Y 420.785,Z 707.31,A -85,B 0,C 180,E1 16408.264,E2 16408.264} C_VEL
LIN {X 0,Y 422.822,Z 712.584,A -85,B 0,C 180,E1 16408.932,E2 16408.932} C_VEL
LIN {X 0,Y 426.03,Z 716.304,A -85,B 0,C 180,E1 16409.789,E2 16409.789} C_VEL
LIN {X 0,Y 443.73,Z 741.829,A -85,B 0,C 180,E1 16414.123,E2 16414.123} C_VEL
LIN {X 0,Y 462.302,Z 772.747,A -85,B 0,C 180,E1 16418.188,E2 16418.188} C_VEL
LIN {X 0,Y 478.627,Z 808.177,A -85,B 0,C 180,E1 16422.008,E2 16422.008} C_VEL
LIN {X 0,Y 483.787,Z 824.121,A -85,B 0,C 180,E1 16423.499,E2 16423.499} C_VEL
LIN {X 0,Y 475.823,Z 867.358,A -85,B 0,C 180,E1 16425.519,E2 16425.519} C_VEL
LIN {X 0,Y 466.161,Z 908.588,A -85,B 0,C 180,E1 16428.254,E2 16428.254} C_VEL
LIN {X 0,Y 455.266,Z 948.442,A -85,B 0,C 180,E1 16431.913,E2 16431.913} C_VEL
LIN {X 0,Y 444.364,Z 985.142,A -85,B 0,C 180,E1 16436.527,E2 16436.527} C_VEL
LIN {X 0,Y 435.08,Z 1016.68,A -85,B 0,C 180,E1 16441.951,E2 16441.951} C_VEL
LIN {X 0,Y 428.547,Z 1041.002,A -85,B 0,C 180,E1 16447.657,E2 16447.657} C_VEL
LIN {X 0,Y 424.522,Z 1060.43,A -85,B 0,C 180,E1 16454.098,E2 16454.098} C_VEL
LIN {X 0,Y 423.05,Z 1071.552,A -85,B 0,C 180,E1 16459.681,E2 16459.681} C_VEL
LIN {X 0,Y 422.682,Z 1076.767,A -85,B 0,C 180,E1 16463.825,E2 16463.825} C_VEL
LIN {X 0,Y 422.738,Z 1079.78,A -85,B 0,C 180,E1 16469.999,E2 16469.999} C_VEL
LIN {X 0,Y 422.663,Z 1076.974,A -85,B 0,C 180,E1 16476.174,E2 16476.174} C_VEL
LIN {X 0,Y 423.176,Z 1070.354,A -85,B 0,C 180,E1 16481.358,E2 16481.358} C_VEL
LIN {X 0,Y 425.383,Z 1056.719,A -85,B 0,C 180,E1 16487.625,E2 16487.625} C_VEL
LIN {X 0,Y 429.787,Z 1037.679,A -85,B 0,C 180,E1 16493.557,E2 16493.557} C_VEL
LIN {X 0,Y 432.023,Z 1029.493,A -85,B 0,C 180,E1 16495.603,E2 16495.603} C_VEL
LIN {X 0,Y 430.744,Z 1021.434,A -85,B 0,C 180,E1 16497.669,E2 16497.669} C_VEL
LIN {X 0,Y 429.713,Z 1012.742,A -85,B 0,C 180,E1 16499.702,E2 16499.702} C_VEL
LIN {X 0,Y 439.819,Z 982.271,A -85,B 0,C 180,E1 16504.855,E2 16504.855} C_VEL
LIN {X 0,Y 451.38,Z 946.266,A -85,B 0,C 180,E1 16509.356,E2 16509.356} C_VEL
LIN {X 0,Y 463.024,Z 906.947,A -85,B 0,C 180,E1 16512.944,E2 16512.944} C_VEL
LIN {X 0,Y 474.017,Z 862.648,A -85,B 0,C 180,E1 16515.832,E2 16515.832} C_VEL
LIN {X 0,Y 480.784,Z 826.324,A -85,B 0,C 180,E1 16517.546,E2 16517.546} C_VEL
LIN {X 0,Y 466.886,Z 792.152,A -85,B 0,C 180,E1 16521.441,E2 16521.441} C_VEL
LIN {X 0,Y 450.122,Z 761.537,A -85,B 0,C 180,E1 16525.678,E2 16525.678} C_VEL
LIN {X 0,Y 432.309,Z 734.738,A -85,B 0,C 180,E1 16530.398,E2 16530.398} C_VEL
LIN {X 0,Y 421.73,Z 720.809,A -85,B 0,C 180,E1 16533.662,E2 16533.662} C_VEL
LIN {X 0,Y 417.075,Z 714.232,A -85,B 0,C 180,E1 16535.305,E2 16535.305} C_VEL
LIN {X 0,Y 413.308,Z 709.355,A -85,B 0,C 180,E1 16536.728,E2 16536.728} C_VEL
LIN {X 0,Y 413.02,Z 707.31,A -85,B 0,C 180,E1 16536.983,E2 16536.983} C_VEL
LIN {X 0,Y 413.278,Z 707.31,A -85,B 0,C 180,E1 16542.946,E2 16542.946} C_VEL
LIN {X 0,Y 413.857,Z 707.31,A -85,B 0,C 180,E1 16549.455,E2 16549.455} C_VEL
LIN {X 0,Y 413.946,Z 707.31,A -85,B 0,C 180,E1 16555.805,E2 16555.805} C_VEL
LIN {X 0,Y 414.222,Z 707.31,A -85,B 0,C 180,E1 16560.004,E2 16560.004} C_VEL
LIN {X 0,Y 413.833,Z 707.31,A -85,B 0,C 180,E1 16566.311,E2 16566.311} C_VEL
LIN {X 0,Y 413.55,Z 707.31,A -85,B 0,C 180,E1 16572.705,E2 16572.705} C_VEL
LIN {X 0,Y 413.218,Z 707.31,A -85,B 0,C 180,E1 16580.126,E2 16580.126} C_VEL
LIN {X 0,Y 413.114,Z 707.467,A -85,B 0,C 180,E1 16581.456,E2 16581.456} C_VEL
LIN {X 0,Y 415.09,Z 712.574,A -85,B 0,C 180,E1 16582.332,E2 16582.332} C_VEL
LIN {X 0,Y 418.543,Z 715.876,A -85,B 0,C 180,E1 16583.545,E2 16583.545} C_VEL
LIN {X 0,Y 433.922,Z 737.254,A -85,B 0,C 180,E1 16588.414,E2 16588.414} C_VEL
LIN {X 0,Y 451.4,Z 764.396,A -85,B 0,C 180,E1 16593.208,E2 16593.208} C_VEL
LIN {X 0,Y 466.571,Z 794.846,A -85,B 0,C 180,E1 16597.447,E2 16597.447} C_VEL
LIN {X 0,Y 478.684,Z 828.008,A -85,B 0,C 180,E1 16601.399,E2 16601.399} C_VEL
LIN {X 0,Y 468.957,Z 871.766,A -85,B 0,C 180,E1 16603.926,E2 16603.926} C_VEL
LIN {X 0,Y 458.175,Z 910.821,A -85,B 0,C 180,E1 16607.078,E2 16607.078} C_VEL
LIN {X 0,Y 447.192,Z 945.751,A -85,B 0,C 180,E1 16610.888,E2 16610.888} C_VEL
LIN {X 0,Y 436.295,Z 978.135,A -85,B 0,C 180,E1 16615.643,E2 16615.643} C_VEL
LIN {X 0,Y 427.039,Z 1005.474,A -85,B 0,C 180,E1 16621.087,E2 16621.087} C_VEL
LIN {X 0,Y 420.432,Z 1027.603,A -85,B 0,C 180,E1 16627.204,E2 16627.204} C_VEL
LIN {X 0,Y 416.6,Z 1043.828,A -85,B 0,C 180,E1 16633.763,E2 16633.763} C_VEL
LIN {X 0,Y 415.087,Z 1052.616,A -85,B 0,C 180,E1 16639.483,E2 16639.483} C_VEL
LIN {X 0,Y 414.539,Z 1057.138,A -85,B 0,C 180,E1 16645.808,E2 16645.808} C_VEL
LIN {X 0,Y 414.86,Z 1057.089,A -85,B 0,C 180,E1 16650.001,E2 16650.001} C_VEL
LIN {X 0,Y 415.083,Z 1052.386,A -85,B 0,C 180,E1 16656.289,E2 16656.289} C_VEL
LIN {X 0,Y 416.511,Z 1043.202,A -85,B 0,C 180,E1 16662.077,E2 16662.077} C_VEL
LIN {X 0,Y 420.071,Z 1027.305,A -85,B 0,C 180,E1 16668.401,E2 16668.401} C_VEL
LIN {X 0,Y 426.62,Z 1004.273,A -85,B 0,C 180,E1 16674.67,E2 16674.67} C_VEL
LIN {X 0,Y 435.789,Z 975.469,A -85,B 0,C 180,E1 16680.28,E2 16680.28} C_VEL
LIN {X 0,Y 446.872,Z 940.71,A -85,B 0,C 180,E1 16685.205,E2 16685.205} C_VEL
LIN {X 0,Y 458.383,Z 901.746,A -85,B 0,C 180,E1 16689.219,E2 16689.219} C_VEL
LIN {X 0,Y 469.04,Z 859.073,A -85,B 0,C 180,E1 16692.396,E2 16692.396} C_VEL
LIN {X 0,Y 475.514,Z 826.587,A -85,B 0,C 180,E1 16694.182,E2 16694.182} C_VEL
LIN {X 0,Y 462.991,Z 791.444,A -85,B 0,C 180,E1 16698.075,E2 16698.075} C_VEL
LIN {X 0,Y 446.403,Z 758.426,A -85,B 0,C 180,E1 16702.331,E2 16702.331} C_VEL
LIN {X 0,Y 428.61,Z 730.973,A -85,B 0,C 180,E1 16706.765,E2 16706.765} C_VEL
LIN {X 0,Y 419.897,Z 719.187,A -85,B 0,C 180,E1 16709.122,E2 16709.122} C_VEL
LIN {X 0,Y 416.367,Z 713.91,A -85,B 0,C 180,E1 16710.175,E2 16710.175} C_VEL
LIN {X 0,Y 412.99,Z 708.988,A -85,B 0,C 180,E1 16711.229,E2 16711.229} C_VEL
LIN {X 0,Y 412.838,Z 707.31,A -85,B 0,C 180,E1 16711.494,E2 16711.494} C_VEL
LIN {X 0,Y 413.056,Z 707.31,A -85,B 0,C 180,E1 16718.473,E2 16718.473} C_VEL
LIN {X 0,Y 413.52,Z 707.31,A -85,B 0,C 180,E1 16725.132,E2 16725.132} C_VEL
LIN {X 0,Y 413.97,Z 707.31,A -85,B 0,C 180,E1 16731.926,E2 16731.926} C_VEL
LIN {X 0,Y 413.938,Z 707.31,A -85,B 0,C 180,E1 16737.898,E2 16737.898} C_VEL
LIN {X 0,Y 414.205,Z 707.31,A -85,B 0,C 180,E1 16742.093,E2 16742.093} C_VEL
LIN {X 0,Y 413.947,Z 707.31,A -85,B 0,C 180,E1 16748.718,E2 16748.718} C_VEL
LIN {X 0,Y 413.461,Z 707.31,A -85,B 0,C 180,E1 16754.862,E2 16754.862} C_VEL
LIN {X 0,Y 413.032,Z 707.31,A -85,B 0,C 180,E1 16761.52,E2 16761.52} C_VEL
LIN {X 0,Y 412.91,Z 707.737,A -85,B 0,C 180,E1 16766.286,E2 16766.286} C_VEL
LIN {X 0,Y 415.176,Z 712.885,A -85,B 0,C 180,E1 16767.067,E2 16767.067} C_VEL
LIN {X 0,Y 418.186,Z 716.213,A -85,B 0,C 180,E1 16767.942,E2 16767.942} C_VEL
LIN {X 0,Y 435.857,Z 741.118,A -85,B 0,C 180,E1 16772.61,E2 16772.61} C_VEL
LIN {X 0,Y 455.009,Z 772.658,A -85,B 0,C 180,E1 16777.052,E2 16777.052} C_VEL
LIN {X 0,Y 470.598,Z 805.94,A -85,B 0,C 180,E1 16780.846,E2 16780.846} C_VEL
LIN {X 0,Y 477.866,Z 826.376,A -85,B 0,C 180,E1 16782.914,E2 16782.914} C_VEL
LIN {X 0,Y 469.711,Z 868.73,A -85,B 0,C 180,E1 16784.939,E2 16784.939} C_VEL
LIN {X 0,Y 459.829,Z 909.322,A -85,B 0,C 180,E1 16787.675,E2 16787.675} C_VEL
LIN {X 0,Y 448.806,Z 948.31,A -85,B 0,C 180,E1 16791.295,E2 16791.295} C_VEL
LIN {X 0,Y 437.924,Z 983.74,A -85,B 0,C 180,E1 16795.783,E2 16795.783} C_VEL
LIN {X 0,Y 428.212,Z 1015.091,A -85,B 0,C 180,E1 16801.171,E2 16801.171} C_VEL
LIN {X 0,Y 421.014,Z 1040.724,A -85,B 0,C 180,E1 16807.235,E2 16807.235} C_VEL
LIN {X 0,Y 416.768,Z 1059.962,A -85,B 0,C 180,E1 16813.71,E2 16813.71} C_VEL
LIN {X 0,Y 415.181,Z 1071.316,A -85,B 0,C 180,E1 16819.484,E2 16819.484} C_VEL
LIN {X 0,Y 414.784,Z 1076.543,A -85,B 0,C 180,E1 16823.707,E2 16823.707} C_VEL
LIN {X 0,Y 414.838,Z 1079.566,A -85,B 0,C 180,E1 16829.999,E2 16829.999} C_VEL
LIN {X 0,Y 414.762,Z 1076.774,A -85,B 0,C 180,E1 16836.292,E2 16836.292} C_VEL
LIN {X 0,Y 415.337,Z 1070.163,A -85,B 0,C 180,E1 16841.575,E2 16841.575} C_VEL
LIN {X 0,Y 417.689,Z 1056.544,A -85,B 0,C 180,E1 16847.961,E2 16847.961} C_VEL
LIN {X 0,Y 422.32,Z 1037.522,A -85,B 0,C 180,E1 16853.999,E2 16853.999} C_VEL
LIN {X 0,Y 429.713,Z 1012.742,A -85,B 0,C 180,E1 16859.702,E2 16859.702} C_VEL
LIN {X 0,Y 429.315,Z 1003.591,A -85,B 0,C 180,E1 16861.701,E2 16861.701} C_VEL
LIN {X 0,Y 429.114,Z 993.863,A -85,B 0,C 180,E1 16863.655,E2 16863.655} C_VEL
LIN {X 0,Y 440.807,Z 959.471,A -85,B 0,C 180,E1 16868.507,E2 16868.507} C_VEL
LIN {X 0,Y 453.285,Z 920.138,A -85,B 0,C 180,E1 16872.542,E2 16872.542} C_VEL
LIN {X 0,Y 464.862,Z 877.969,A -85,B 0,C 180,E1 16875.647,E2 16875.647} C_VEL
LIN {X 0,Y 475.077,Z 831.861,A -85,B 0,C 180,E1 16877.968,E2 16877.968} C_VEL
LIN {X 0,Y 467.173,Z 808.496,A -85,B 0,C 180,E1 16880.529,E2 16880.529} C_VEL
LIN {X 0,Y 451.28,Z 775.669,A -85,B 0,C 180,E1 16884.873,E2 16884.873} C_VEL
LIN {X 0,Y 433.52,Z 747.198,A -85,B 0,C 180,E1 16889.695,E2 16889.695} C_VEL
LIN {X 0,Y 419.492,Z 727.901,A -85,B 0,C 180,E1 16894.027,E2 16894.027} C_VEL
LIN {X 0,Y 414.228,Z 721.018,A -85,B 0,C 180,E1 16895.916,E2 16895.916} C_VEL
LIN {X 0,Y 409.73,Z 714.511,A -85,B 0,C 180,E1 16897.726,E2 16897.726} C_VEL
LIN {X 0,Y 405.56,Z 709.888,A -85,B 0,C 180,E1 16899.513,E2 16899.513} C_VEL
LIN {X 0,Y 405.134,Z 707.31,A -85,B 0,C 180,E1 16899.851,E2 16899.851} C_VEL
LIN {X 0,Y 405.683,Z 707.31,A -85,B 0,C 180,E1 16907.053,E2 16907.053} C_VEL
LIN {X 0,Y 406.046,Z 707.31,A -85,B 0,C 180,E1 16913.576,E2 16913.576} C_VEL
LIN {X 0,Y 406.317,Z 707.31,A -85,B 0,C 180,E1 16920.004,E2 16920.004} C_VEL
LIN {X 0,Y 405.909,Z 707.31,A -85,B 0,C 180,E1 16926.434,E2 16926.434} C_VEL
LIN {X 0,Y 405.545,Z 707.31,A -85,B 0,C 180,E1 16933.706,E2 16933.706} C_VEL
LIN {X 0,Y 405.314,Z 707.586,A -85,B 0,C 180,E1 16938.604,E2 16938.604} C_VEL
LIN {X 0,Y 407.312,Z 712.565,A -85,B 0,C 180,E1 16939.631,E2 16939.631} C_VEL
LIN {X 0,Y 410.943,Z 715.974,A -85,B 0,C 180,E1 16941.1,E2 16941.1} C_VEL
LIN {X 0,Y 415.329,Z 721.722,A -85,B 0,C 180,E1 16942.797,E2 16942.797} C_VEL
LIN {X 0,Y 431.098,Z 744.009,A -85,B 0,C 180,E1 16948.01,E2 16948.01} C_VEL
LIN {X 0,Y 447.644,Z 770.581,A -85,B 0,C 180,E1 16952.799,E2 16952.799} C_VEL
LIN {X 0,Y 462.015,Z 800.486,A -85,B 0,C 180,E1 16957.065,E2 16957.065} C_VEL
LIN {X 0,Y 472.661,Z 830.765,A -85,B 0,C 180,E1 16960.784,E2 16960.784} C_VEL
LIN {X 0,Y 462.349,Z 875.912,A -85,B 0,C 180,E1 16963.5,E2 16963.5} C_VEL
LIN {X 0,Y 450.563,Z 916.439,A -85,B 0,C 180,E1 16966.908,E2 16966.908} C_VEL
LIN {X 0,Y 438.261,Z 953.463,A -85,B 0,C 180,E1 16971.213,E2 16971.213} C_VEL
LIN {X 0,Y 426.803,Z 985.941,A -85,B 0,C 180,E1 16976.404,E2 16976.404} C_VEL
LIN {X 0,Y 417.575,Z 1012.94,A -85,B 0,C 180,E1 16982.385,E2 16982.385} C_VEL
LIN {X 0,Y 411.344,Z 1033.417,A -85,B 0,C 180,E1 16988.798,E2 16988.798} C_VEL
LIN {X 0,Y 408.33,Z 1046.646,A -85,B 0,C 180,E1 16994.944,E2 16994.944} C_VEL
LIN {X 0,Y 407.045,Z 1053.905,A -85,B 0,C 180,E1 17000.278,E2 17000.278} C_VEL
LIN {X 0,Y 406.634,Z 1057.345,A -85,B 0,C 180,E1 17005.727,E2 17005.727} C_VEL
LIN {X 0,Y 406.975,Z 1057.304,A -85,B 0,C 180,E1 17010.001,E2 17010.001} C_VEL
LIN {X 0,Y 407.211,Z 1052.624,A -85,B 0,C 180,E1 17016.411,E2 17016.411} C_VEL
LIN {X 0,Y 408.716,Z 1043.466,A -85,B 0,C 180,E1 17022.311,E2 17022.311} C_VEL
LIN {X 0,Y 412.47,Z 1027.593,A -85,B 0,C 180,E1 17028.753,E2 17028.753} C_VEL
LIN {X 0,Y 419.205,Z 1005.017,A -85,B 0,C 180,E1 17035.028,E2 17035.028} C_VEL
LIN {X 0,Y 428.873,Z 975.821,A -85,B 0,C 180,E1 17040.822,E2 17040.822} C_VEL
LIN {X 0,Y 440.37,Z 941.103,A -85,B 0,C 180,E1 17045.804,E2 17045.804} C_VEL
LIN {X 0,Y 452.257,Z 902.193,A -85,B 0,C 180,E1 17049.855,E2 17049.855} C_VEL
LIN {X 0,Y 463.162,Z 859.915,A -85,B 0,C 180,E1 17053.037,E2 17053.037} C_VEL
LIN {X 0,Y 469.476,Z 829.444,A -85,B 0,C 180,E1 17054.751,E2 17054.751} C_VEL
LIN {X 0,Y 457.318,Z 794.676,A -85,B 0,C 180,E1 17058.736,E2 17058.736} C_VEL
LIN {X 0,Y 441.519,Z 762.657,A -85,B 0,C 180,E1 17063.022,E2 17063.022} C_VEL
LIN {X 0,Y 423.359,Z 733.983,A -85,B 0,C 180,E1 17067.825,E2 17067.825} C_VEL
LIN {X 0,Y 412.955,Z 720.187,A -85,B 0,C 180,E1 17070.828,E2 17070.828} C_VEL
LIN {X 0,Y 408.811,Z 714.087,A -85,B 0,C 180,E1 17072.179,E2 17072.179} C_VEL
LIN {X 0,Y 405.202,Z 709.237,A -85,B 0,C 180,E1 17073.415,E2 17073.415} C_VEL
LIN {X 0,Y 404.985,Z 707.31,A -85,B 0,C 180,E1 17073.654,E2 17073.654} C_VEL
LIN {X 0,Y 405.213,Z 707.31,A -85,B 0,C 180,E1 17080.328,E2 17080.328} C_VEL
LIN {X 0,Y 405.786,Z 707.31,A -85,B 0,C 180,E1 17087.048,E2 17087.048} C_VEL
LIN {X 0,Y 406.225,Z 707.31,A -85,B 0,C 180,E1 17093.571,E2 17093.571} C_VEL
LIN {X 0,Y 406.334,Z 707.31,A -85,B 0,C 180,E1 17099.996,E2 17099.996} C_VEL
LIN {X 0,Y 406.06,Z 707.31,A -85,B 0,C 180,E1 17106.424,E2 17106.424} C_VEL
LIN {X 0,Y 405.696,Z 707.31,A -85,B 0,C 180,E1 17112.947,E2 17112.947} C_VEL
LIN {X 0,Y 405.177,Z 707.31,A -85,B 0,C 180,E1 17119.666,E2 17119.666} C_VEL
LIN {X 0,Y 405.07,Z 708.064,A -85,B 0,C 180,E1 17124.08,E2 17124.08} C_VEL
LIN {X 0,Y 407.613,Z 713.205,A -85,B 0,C 180,E1 17125.03,E2 17125.03} C_VEL
LIN {X 0,Y 410.506,Z 716.388,A -85,B 0,C 180,E1 17125.96,E2 17125.96} C_VEL
LIN {X 0,Y 425.65,Z 737.479,A -85,B 0,C 180,E1 17130.379,E2 17130.379} C_VEL
LIN {X 0,Y 443.559,Z 765.145,A -85,B 0,C 180,E1 17134.821,E2 17134.821} C_VEL
LIN {X 0,Y 460.634,Z 798.66,A -85,B 0,C 180,E1 17139.06,E2 17139.06} C_VEL
LIN {X 0,Y 471.815,Z 828.482,A -85,B 0,C 180,E1 17142.281,E2 17142.281} C_VEL
LIN {X 0,Y 462.804,Z 873.761,A -85,B 0,C 180,E1 17144.555,E2 17144.555} C_VEL
LIN {X 0,Y 452.564,Z 913.562,A -85,B 0,C 180,E1 17147.37,E2 17147.37} C_VEL
LIN {X 0,Y 441.638,Z 950.556,A -85,B 0,C 180,E1 17150.932,E2 17150.932} C_VEL
LIN {X 0,Y 430.638,Z 985.119,A -85,B 0,C 180,E1 17155.428,E2 17155.428} C_VEL
LIN {X 0,Y 420.643,Z 1016.089,A -85,B 0,C 180,E1 17160.898,E2 17160.898} C_VEL
LIN {X 0,Y 413.473,Z 1040.445,A -85,B 0,C 180,E1 17166.796,E2 17166.796} C_VEL
LIN {X 0,Y 409.053,Z 1059.433,A -85,B 0,C 180,E1 17173.284,E2 17173.284} C_VEL
LIN {X 0,Y 407.308,Z 1071.079,A -85,B 0,C 180,E1 17179.278,E2 17179.278} C_VEL
LIN {X 0,Y 406.917,Z 1076.319,A -85,B 0,C 180,E1 17183.584,E2 17183.584} C_VEL
LIN {X 0,Y 406.952,Z 1079.353,A -85,B 0,C 180,E1 17189.999,E2 17189.999} C_VEL
LIN {X 0,Y 406.894,Z 1076.575,A -85,B 0,C 180,E1 17196.414,E2 17196.414} C_VEL
LIN {X 0,Y 407.479,Z 1069.972,A -85,B 0,C 180,E1 17201.802,E2 17201.802} C_VEL
LIN {X 0,Y 409.961,Z 1056.368,A -85,B 0,C 180,E1 17208.311,E2 17208.311} C_VEL
LIN {X 0,Y 414.625,Z 1038.236,A -85,B 0,C 180,E1 17214.219,E2 17214.219} C_VEL
LIN {X 0,Y 422.274,Z 1013.743,A -85,B 0,C 180,E1 17220.027,E2 17220.027} C_VEL
LIN {X 0,Y 429.114,Z 993.863,A -85,B 0,C 180,E1 17223.655,E2 17223.655} C_VEL
LIN {X 0,Y 429.282,Z 983.707,A -85,B 0,C 180,E1 17225.559,E2 17225.559} C_VEL
LIN {X 0,Y 429.735,Z 972.973,A -85,B 0,C 180,E1 17227.417,E2 17227.417} C_VEL
LIN {X 0,Y 442.788,Z 934.841,A -85,B 0,C 180,E1 17231.863,E2 17231.863} C_VEL
LIN {X 0,Y 455.164,Z 893.693,A -85,B 0,C 180,E1 17235.312,E2 17235.312} C_VEL
LIN {X 0,Y 465.955,Z 850.189,A -85,B 0,C 180,E1 17237.876,E2 17237.876} C_VEL
LIN {X 0,Y 469.073,Z 832.414,A -85,B 0,C 180,E1 17238.757,E2 17238.757} C_VEL
LIN {X 0,Y 456.213,Z 799.281,A -85,B 0,C 180,E1 17242.816,E2 17242.816} C_VEL
LIN {X 0,Y 440.858,Z 770.198,A -85,B 0,C 180,E1 17247.153,E2 17247.153} C_VEL
LIN {X 0,Y 425.457,Z 746.44,A -85,B 0,C 180,E1 17251.7,E2 17251.7} C_VEL
LIN {X 0,Y 412.626,Z 728.633,A -85,B 0,C 180,E1 17256.105,E2 17256.105} C_VEL
LIN {X 0,Y 406.979,Z 721.435,A -85,B 0,C 180,E1 17258.393,E2 17258.393} C_VEL
LIN {X 0,Y 403.162,Z 715.83,A -85,B 0,C 180,E1 17260.167,E2 17260.167} C_VEL
LIN {X 0,Y 397.808,Z 709.733,A -85,B 0,C 180,E1 17262.926,E2 17262.926} C_VEL
LIN {X 0,Y 397.439,Z 707.31,A -85,B 0,C 180,E1 17263.388,E2 17263.388} C_VEL
LIN {X 0,Y 397.966,Z 707.31,A -85,B 0,C 180,E1 17269.028,E2 17269.028} C_VEL
LIN {X 0,Y 398.126,Z 707.31,A -85,B 0,C 180,E1 17275.638,E2 17275.638} C_VEL
LIN {X 0,Y 398.412,Z 707.31,A -85,B 0,C 180,E1 17280.004,E2 17280.004} C_VEL
LIN {X 0,Y 397.987,Z 707.31,A -85,B 0,C 180,E1 17286.563,E2 17286.563} C_VEL
LIN {X 0,Y 397.617,Z 707.31,A -85,B 0,C 180,E1 17293.985,E2 17293.985} C_VEL
LIN {X 0,Y 397.628,Z 707.81,A -85,B 0,C 180,E1 17295.196,E2 17295.196} C_VEL
LIN {X 0,Y 399.625,Z 712.749,A -85,B 0,C 180,E1 17296.456,E2 17296.456} C_VEL
LIN {X 0,Y 403.393,Z 716.016,A -85,B 0,C 180,E1 17298.271,E2 17298.271} C_VEL
LIN {X 0,Y 407.713,Z 721.783,A -85,B 0,C 180,E1 17300.227,E2 17300.227} C_VEL
LIN {X 0,Y 419.606,Z 738.242,A -85,B 0,C 180,E1 17304.757,E2 17304.757} C_VEL
LIN {X 0,Y 434.794,Z 760.828,A -85,B 0,C 180,E1 17309.637,E2 17309.637} C_VEL
LIN {X 0,Y 451.004,Z 791.167,A -85,B 0,C 180,E1 17314.619,E2 17314.619} C_VEL
LIN {X 0,Y 463.523,Z 823.249,A -85,B 0,C 180,E1 17318.91,E2 17318.91} C_VEL
LIN {X 0,Y 466.715,Z 835.424,A -85,B 0,C 180,E1 17320.333,E2 17320.333} C_VEL
LIN {X 0,Y 456.372,Z 877.492,A -85,B 0,C 180,E1 17322.888,E2 17322.888} C_VEL
LIN {X 0,Y 444.534,Z 916.919,A -85,B 0,C 180,E1 17326.242,E2 17326.242} C_VEL
LIN {X 0,Y 431.98,Z 953.378,A -85,B 0,C 180,E1 17330.518,E2 17330.518} C_VEL
LIN {X 0,Y 420.068,Z 985.885,A -85,B 0,C 180,E1 17335.761,E2 17335.761} C_VEL
LIN {X 0,Y 410.422,Z 1012.777,A -85,B 0,C 180,E1 17341.782,E2 17341.782} C_VEL
LIN {X 0,Y 403.654,Z 1033.975,A -85,B 0,C 180,E1 17348.53,E2 17348.53} C_VEL
LIN {X 0,Y 400.539,Z 1046.818,A -85,B 0,C 180,E1 17354.644,E2 17354.644} C_VEL
LIN {X 0,Y 399.096,Z 1054.811,A -85,B 0,C 180,E1 17360.858,E2 17360.858} C_VEL
LIN {X 0,Y 398.729,Z 1057.553,A -85,B 0,C 180,E1 17365.642,E2 17365.642} C_VEL
LIN {X 0,Y 399.073,Z 1057.518,A -85,B 0,C 180,E1 17370.001,E2 17370.001} C_VEL
LIN {X 0,Y 399.331,Z 1052.862,A -85,B 0,C 180,E1 17376.538,E2 17376.538} C_VEL
LIN {X 0,Y 400.917,Z 1043.729,A -85,B 0,C 180,E1 17382.554,E2 17382.554} C_VEL
LIN {X 0,Y 404.874,Z 1027.879,A -85,B 0,C 180,E1 17389.118,E2 17389.118} C_VEL
LIN {X 0,Y 411.705,Z 1005.965,A -85,B 0,C 180,E1 17395.342,E2 17395.342} C_VEL
LIN {X 0,Y 421.473,Z 977.622,A -85,B 0,C 180,E1 17401.122,E2 17401.122} C_VEL
LIN {X 0,Y 432.588,Z 945.345,A -85,B 0,C 180,E1 17405.929,E2 17405.929} C_VEL
LIN {X 0,Y 444.054,Z 909.577,A -85,B 0,C 180,E1 17409.863,E2 17409.863} C_VEL
LIN {X 0,Y 454.826,Z 870.637,A -85,B 0,C 180,E1 17413.031,E2 17413.031} C_VEL
LIN {X 0,Y 463.437,Z 832.441,A -85,B 0,C 180,E1 17415.309,E2 17415.309} C_VEL
LIN {X 0,Y 452.37,Z 799.561,A -85,B 0,C 180,E1 17419.21,E2 17419.21} C_VEL
LIN {X 0,Y 437.508,Z 768.462,A -85,B 0,C 180,E1 17423.498,E2 17423.498} C_VEL
LIN {X 0,Y 420.599,Z 740.903,A -85,B 0,C 180,E1 17428.198,E2 17428.198} C_VEL
LIN {X 0,Y 406.001,Z 720.927,A -85,B 0,C 180,E1 17432.712,E2 17432.712} C_VEL
LIN {X 0,Y 401.09,Z 714.171,A -85,B 0,C 180,E1 17434.475,E2 17434.475} C_VEL
LIN {X 0,Y 397.375,Z 709.274,A -85,B 0,C 180,E1 17435.914,E2 17435.914} C_VEL
LIN {X 0,Y 397.105,Z 707.31,A -85,B 0,C 180,E1 17436.157,E2 17436.157} C_VEL
LIN {X 0,Y 397.473,Z 707.31,A -85,B 0,C 180,E1 17442.395,E2 17442.395} C_VEL
LIN {X 0,Y 398.044,Z 707.31,A -85,B 0,C 180,E1 17449.023,E2 17449.023} C_VEL
LIN {X 0,Y 398.254,Z 707.31,A -85,B 0,C 180,E1 17455.632,E2 17455.632} C_VEL
LIN {X 0,Y 398.401,Z 707.31,A -85,B 0,C 180,E1 17462.176,E2 17462.176} C_VEL
LIN {X 0,Y 398.147,Z 707.31,A -85,B 0,C 180,E1 17468.753,E2 17468.753} C_VEL
LIN {X 0,Y 397.553,Z 707.31,A -85,B 0,C 180,E1 17475.471,E2 17475.471} C_VEL
LIN {X 0,Y 397.222,Z 708.035,A -85,B 0,C 180,E1 17481.559,E2 17481.559} C_VEL
LIN {X 0,Y 399.922,Z 713.267,A -85,B 0,C 180,E1 17482.694,E2 17482.694} C_VEL
LIN {X 0,Y 402.553,Z 715.706,A -85,B 0,C 180,E1 17483.629,E2 17483.629} C_VEL
LIN {X 0,Y 406.838,Z 721.529,A -85,B 0,C 180,E1 17485.134,E2 17485.134} C_VEL
LIN {X 0,Y 425.196,Z 747.383,A -85,B 0,C 180,E1 17490.594,E2 17490.594} C_VEL
LIN {X 0,Y 443.529,Z 778.028,A -85,B 0,C 180,E1 17495.356,E2 17495.356} C_VEL
LIN {X 0,Y 458.972,Z 811.651,A -85,B 0,C 180,E1 17499.534,E2 17499.534} C_VEL
LIN {X 0,Y 465.738,Z 832.826,A -85,B 0,C 180,E1 17501.772,E2 17501.772} C_VEL
LIN {X 0,Y 455.879,Z 878.611,A -85,B 0,C 180,E1 17504.148,E2 17504.148} C_VEL
LIN {X 0,Y 444.415,Z 921.046,A -85,B 0,C 180,E1 17507.334,E2 17507.334} C_VEL
LIN {X 0,Y 432.376,Z 959.509,A -85,B 0,C 180,E1 17511.346,E2 17511.346} C_VEL
LIN {X 0,Y 420.401,Z 994.903,A -85,B 0,C 180,E1 17516.411,E2 17516.411} C_VEL
LIN {X 0,Y 410.643,Z 1024.729,A -85,B 0,C 180,E1 17522.325,E2 17522.325} C_VEL
LIN {X 0,Y 404.01,Z 1047.334,A -85,B 0,C 180,E1 17528.548,E2 17528.548} C_VEL
LIN {X 0,Y 400.467,Z 1064.085,A -85,B 0,C 180,E1 17535.2,E2 17535.2} C_VEL
LIN {X 0,Y 399.142,Z 1073.793,A -85,B 0,C 180,E1 17541.264,E2 17541.264} C_VEL
LIN {X 0,Y 398.894,Z 1078.786,A -85,B 0,C 180,E1 17547.822,E2 17547.822} C_VEL
LIN {X 0,Y 398.995,Z 1078.842,A -85,B 0,C 180,E1 17552.176,E2 17552.176} C_VEL
LIN {X 0,Y 399.085,Z 1074.198,A -85,B 0,C 180,E1 17558.735,E2 17558.735} C_VEL
LIN {X 0,Y 400.467,Z 1064.924,A -85,B 0,C 180,E1 17564.798,E2 17564.798} C_VEL
LIN {X 0,Y 404.2,Z 1048.768,A -85,B 0,C 180,E1 17571.403,E2 17571.403} C_VEL
LIN {X 0,Y 411.049,Z 1026.205,A -85,B 0,C 180,E1 17577.783,E2 17577.783} C_VEL
LIN {X 0,Y 420.648,Z 998.506,A -85,B 0,C 180,E1 17583.443,E2 17583.443} C_VEL
LIN {X 0,Y 429.735,Z 972.973,A -85,B 0,C 180,E1 17587.417,E2 17587.417} C_VEL
LIN {X 0,Y 430.38,Z 961.788,A -85,B 0,C 180,E1 17589.219,E2 17589.219} C_VEL
LIN {X 0,Y 431.492,Z 950.053,A -85,B 0,C 180,E1 17590.944,E2 17590.944} C_VEL
LIN {X 0,Y 444.035,Z 912.072,A -85,B 0,C 180,E1 17594.626,E2 17594.626} C_VEL
LIN {X 0,Y 455.296,Z 872.297,A -85,B 0,C 180,E1 17597.425,E2 17597.425} C_VEL
LIN {X 0,Y 463.454,Z 836.185,A -85,B 0,C 180,E1 17599.284,E2 17599.284} C_VEL
LIN {X 0,Y 451.305,Z 803.831,A -85,B 0,C 180,E1 17603.377,E2 17603.377} C_VEL
LIN {X 0,Y 436.249,Z 774.599,A -85,B 0,C 180,E1 17607.914,E2 17607.914} C_VEL
LIN {X 0,Y 420.549,Z 749.533,A -85,B 0,C 180,E1 17612.872,E2 17612.872} C_VEL
LIN {X 0,Y 409.224,Z 734.522,A -85,B 0,C 180,E1 17616.979,E2 17616.979} C_VEL
LIN {X 0,Y 404.947,Z 728.647,A -85,B 0,C 180,E1 17618.8,E2 17618.8} C_VEL
LIN {X 0,Y 399.863,Z 721.858,A -85,B 0,C 180,E1 17621.241,E2 17621.241} C_VEL
LIN {X 0,Y 395.882,Z 716.41,A -85,B 0,C 180,E1 17623.467,E2 17623.467} C_VEL
LIN {X 0,Y 394.365,Z 714.519,A -85,B 0,C 180,E1 17624.401,E2 17624.401} C_VEL
LIN {X 0,Y 390.316,Z 709.884,A -85,B 0,C 180,E1 17627.247,E2 17627.247} C_VEL
LIN {X 0,Y 389.902,Z 707.31,A -85,B 0,C 180,E1 17627.946,E2 17627.946} C_VEL
LIN {X 0,Y 390.238,Z 707.31,A -85,B 0,C 180,E1 17633.314,E2 17633.314} C_VEL
LIN {X 0,Y 390.507,Z 707.31,A -85,B 0,C 180,E1 17640.004,E2 17640.004} C_VEL
LIN {X 0,Y 390.091,Z 707.31,A -85,B 0,C 180,E1 17646.697,E2 17646.697} C_VEL
LIN {X 0,Y 389.914,Z 708.086,A -85,B 0,C 180,E1 17650.642,E2 17650.642} C_VEL
LIN {X 0,Y 392.185,Z 712.987,A -85,B 0,C 180,E1 17652.557,E2 17652.557} C_VEL
LIN {X 0,Y 395.88,Z 715.953,A -85,B 0,C 180,E1 17654.836,E2 17654.836} C_VEL
LIN {X 0,Y 399.461,Z 721.476,A -85,B 0,C 180,E1 17656.892,E2 17656.892} C_VEL
LIN {X 0,Y 401.826,Z 724.15,A -85,B 0,C 180,E1 17658.06,E2 17658.06} C_VEL
LIN {X 0,Y 407.567,Z 732.004,A -85,B 0,C 180,E1 17660.66,E2 17660.66} C_VEL
LIN {X 0,Y 417.238,Z 745.358,A -85,B 0,C 180,E1 17664.406,E2 17664.406} C_VEL
LIN {X 0,Y 431.542,Z 767.403,A -85,B 0,C 180,E1 17669.231,E2 17669.231} C_VEL
LIN {X 0,Y 446.965,Z 797.479,A -85,B 0,C 180,E1 17674.289,E2 17674.289} C_VEL
LIN {X 0,Y 458.411,Z 828.406,A -85,B 0,C 180,E1 17678.527,E2 17678.527} C_VEL
LIN {X 0,Y 460.867,Z 838.274,A -85,B 0,C 180,E1 17679.726,E2 17679.726} C_VEL
LIN {X 0,Y 450.237,Z 879.807,A -85,B 0,C 180,E1 17682.315,E2 17682.315} C_VEL
LIN {X 0,Y 438.453,Z 917.723,A -85,B 0,C 180,E1 17685.592,E2 17685.592} C_VEL
LIN {X 0,Y 425.026,Z 955.285,A -85,B 0,C 180,E1 17690.077,E2 17690.077} C_VEL
LIN {X 0,Y 412.978,Z 986.94,A -85,B 0,C 180,E1 17695.304,E2 17695.304} C_VEL
LIN {X 0,Y 402.87,Z 1013.903,A -85,B 0,C 180,E1 17701.499,E2 17701.499} C_VEL
LIN {X 0,Y 396.099,Z 1034.125,A -85,B 0,C 180,E1 17708.099,E2 17708.099} C_VEL
LIN {X 0,Y 392.603,Z 1047.779,A -85,B 0,C 180,E1 17714.802,E2 17714.802} C_VEL
LIN {X 0,Y 391.18,Z 1055.315,A -85,B 0,C 180,E1 17721.087,E2 17721.087} C_VEL
LIN {X 0,Y 390.869,Z 1058.078,A -85,B 0,C 180,E1 17727.779,E2 17727.779} C_VEL
LIN {X 0,Y 391.134,Z 1056.79,A -85,B 0,C 180,E1 17732.221,E2 17732.221} C_VEL
LIN {X 0,Y 391.65,Z 1051.864,A -85,B 0,C 180,E1 17737.784,E2 17737.784} C_VEL
LIN {X 0,Y 393.922,Z 1040.62,A -85,B 0,C 180,E1 17744.482,E2 17744.482} C_VEL
LIN {X 0,Y 398.857,Z 1022.868,A -85,B 0,C 180,E1 17751.228,E2 17751.228} C_VEL
LIN {X 0,Y 406.417,Z 1000.505,A -85,B 0,C 180,E1 17757.18,E2 17757.18} C_VEL
LIN {X 0,Y 416.266,Z 973.374,A -85,B 0,C 180,E1 17762.479,E2 17762.479} C_VEL
LIN {X 0,Y 427.855,Z 940.825,A -85,B 0,C 180,E1 17767.185,E2 17767.185} C_VEL
LIN {X 0,Y 440.157,Z 903.085,A -85,B 0,C 180,E1 17771.183,E2 17771.183} C_VEL
LIN {X 0,Y 451.818,Z 860.606,A -85,B 0,C 180,E1 17774.427,E2 17774.427} C_VEL
LIN {X 0,Y 457.371,Z 835.202,A -85,B 0,C 180,E1 17775.906,E2 17775.906} C_VEL
LIN {X 0,Y 446.741,Z 802.977,A -85,B 0,C 180,E1 17779.868,E2 17779.868} C_VEL
LIN {X 0,Y 433.291,Z 774.107,A -85,B 0,C 180,E1 17783.985,E2 17783.985} C_VEL
LIN {X 0,Y 417.415,Z 747.327,A -85,B 0,C 180,E1 17788.69,E2 17788.69} C_VEL
LIN {X 0,Y 403.586,Z 727.929,A -85,B 0,C 180,E1 17793.14,E2 17793.14} C_VEL
LIN {X 0,Y 398.241,Z 720.932,A -85,B 0,C 180,E1 17795.101,E2 17795.101} C_VEL
LIN {X 0,Y 393.528,Z 714.351,A -85,B 0,C 180,E1 17797.037,E2 17797.037} C_VEL
LIN {X 0,Y 389.609,Z 709.686,A -85,B 0,C 180,E1 17798.779,E2 17798.779} C_VEL
LIN {X 0,Y 389.302,Z 707.31,A -85,B 0,C 180,E1 17799.106,E2 17799.106} C_VEL
LIN {X 0,Y 389.896,Z 707.31,A -85,B 0,C 180,E1 17806.51,E2 17806.51} C_VEL
LIN {X 0,Y 390.389,Z 707.31,A -85,B 0,C 180,E1 17813.309,E2 17813.309} C_VEL
LIN {X 0,Y 390.524,Z 707.31,A -85,B 0,C 180,E1 17819.996,E2 17819.996} C_VEL
LIN {X 0,Y 390.252,Z 707.31,A -85,B 0,C 180,E1 17826.686,E2 17826.686} C_VEL
LIN {X 0,Y 389.807,Z 707.31,A -85,B 0,C 180,E1 17833.613,E2 17833.613} C_VEL
LIN {X 0,Y 389.437,Z 708.053,A -85,B 0,C 180,E1 17838.647,E2 17838.647} C_VEL
LIN {X 0,Y 391.832,Z 713.049,A -85,B 0,C 180,E1 17839.849,E2 17839.849} C_VEL
LIN {X 0,Y 395.058,Z 716.076,A -85,B 0,C 180,E1 17841.177,E2 17841.177} C_VEL
LIN {X 0,Y 399.702,Z 721.88,A -85,B 0,C 180,E1 17842.996,E2 17842.996} C_VEL
LIN {X 0,Y 415.872,Z 744.948,A -85,B 0,C 180,E1 17848.366,E2 17848.366} C_VEL
LIN {X 0,Y 432.631,Z 771.32,A -85,B 0,C 180,E1 17853.062,E2 17853.062} C_VEL
LIN {X 0,Y 448.465,Z 803.067,A -85,B 0,C 180,E1 17857.457,E2 17857.457} C_VEL
LIN {X 0,Y 459.894,Z 834.904,A -85,B 0,C 180,E1 17861.142,E2 17861.142} C_VEL
LIN {X 0,Y 449.781,Z 880.08,A -85,B 0,C 180,E1 17863.537,E2 17863.537} C_VEL
LIN {X 0,Y 437.887,Z 922.496,A -85,B 0,C 180,E1 17866.784,E2 17866.784} C_VEL
LIN {X 0,Y 425.643,Z 960.353,A -85,B 0,C 180,E1 17870.806,E2 17870.806} C_VEL
LIN {X 0,Y 413.421,Z 995.118,A -85,B 0,C 180,E1 17875.875,E2 17875.875} C_VEL
LIN {X 0,Y 403.189,Z 1025.089,A -85,B 0,C 180,E1 17881.946,E2 17881.946} C_VEL
LIN {X 0,Y 396.472,Z 1047.061,A -85,B 0,C 180,E1 17888.119,E2 17888.119} C_VEL
LIN {X 0,Y 392.722,Z 1063.437,A -85,B 0,C 180,E1 17894.708,E2 17894.708} C_VEL
LIN {X 0,Y 391.268,Z 1073.562,A -85,B 0,C 180,E1 17901.087,E2 17901.087} C_VEL
LIN {X 0,Y 390.999,Z 1078.572,A -85,B 0,C 180,E1 17907.778,E2 17907.778} C_VEL
LIN {X 0,Y 391.112,Z 1078.634,A -85,B 0,C 180,E1 17912.219,E2 17912.219} C_VEL
LIN {X 0,Y 391.216,Z 1074.003,A -85,B 0,C 180,E1 17918.912,E2 17918.912} C_VEL
LIN {X 0,Y 392.8,Z 1064.255,A -85,B 0,C 180,E1 17925.334,E2 17925.334} C_VEL
LIN {X 0,Y 396.666,Z 1048.5,A -85,B 0,C 180,E1 17931.868,E2 17931.868} C_VEL
LIN {X 0,Y 404.32,Z 1024.813,A -85,B 0,C 180,E1 17938.633,E2 17938.633} C_VEL
LIN {X 0,Y 414.886,Z 995.643,A -85,B 0,C 180,E1 17944.561,E2 17944.561} C_VEL
LIN {X 0,Y 427.597,Z 961.094,A -85,B 0,C 180,E1 17949.635,E2 17949.635} C_VEL
LIN {X 0,Y 431.492,Z 950.053,A -85,B 0,C 180,E1 17950.944,E2 17950.944} C_VEL
LIN {X 0,Y 432.787,Z 937.889,A -85,B 0,C 180,E1 17952.61,E2 17952.61} C_VEL
LIN {X 0,Y 434.024,Z 925.236,A -85,B 0,C 180,E1 17954.208,E2 17954.208} C_VEL
LIN {X 0,Y 446.17,Z 886.158,A -85,B 0,C 180,E1 17957.295,E2 17957.295} C_VEL
LIN {X 0,Y 456.831,Z 844.469,A -85,B 0,C 180,E1 17959.637,E2 17959.637} C_VEL
LIN {X 0,Y 457.357,Z 838.148,A -85,B 0,C 180,E1 17960.04,E2 17960.04} C_VEL
LIN {X 0,Y 445.297,Z 805.914,A -85,B 0,C 180,E1 17964.315,E2 17964.315} C_VEL
LIN {X 0,Y 430.806,Z 777.364,A -85,B 0,C 180,E1 17968.979,E2 17968.979} C_VEL
LIN {X 0,Y 416.555,Z 754.739,A -85,B 0,C 180,E1 17973.758,E2 17973.758} C_VEL
LIN {X 0,Y 403.827,Z 736.574,A -85,B 0,C 180,E1 17978.831,E2 17978.831} C_VEL
LIN {X 0,Y 397.797,Z 729.077,A -85,B 0,C 180,E1 17981.752,E2 17981.752} C_VEL
LIN {X 0,Y 392.975,Z 722.208,A -85,B 0,C 180,E1 17984.631,E2 17984.631} C_VEL
LIN {X 0,Y 388.848,Z 717.172,A -85,B 0,C 180,E1 17987.639,E2 17987.639} C_VEL
LIN {X 0,Y 388.026,Z 714.969,A -85,B 0,C 180,E1 17988.461,E2 17988.461} C_VEL
LIN {X 0,Y 382.434,Z 708.204,A -85,B 0,C 180,E1 17996.739,E2 17996.739} C_VEL
LIN {X 0,Y 382.387,Z 707.637,A -85,B 0,C 180,E1 18001.139,E2 18001.139} C_VEL
LIN {X 0,Y 387.014,Z 714.636,A -85,B 0,C 180,E1 18009.015,E2 18009.015} C_VEL
LIN {X 0,Y 388.557,Z 716.233,A -85,B 0,C 180,E1 18010.396,E2 18010.396} C_VEL
LIN {X 0,Y 392.022,Z 721.575,A -85,B 0,C 180,E1 18013.11,E2 18013.11} C_VEL
LIN {X 0,Y 394.315,Z 723.784,A -85,B 0,C 180,E1 18014.541,E2 18014.541} C_VEL
LIN {X 0,Y 398.763,Z 729.586,A -85,B 0,C 180,E1 18017.047,E2 18017.047} C_VEL
LIN {X 0,Y 410.003,Z 745.275,A -85,B 0,C 180,E1 18022.165,E2 18022.165} C_VEL
LIN {X 0,Y 423.379,Z 765.909,A -85,B 0,C 180,E1 18027.178,E2 18027.178} C_VEL
LIN {X 0,Y 436.988,Z 791.157,A -85,B 0,C 180,E1 18031.931,E2 18031.931} C_VEL
LIN {X 0,Y 448.561,Z 818.897,A -85,B 0,C 180,E1 18036.165,E2 18036.165} C_VEL
LIN {X 0,Y 455.122,Z 841.028,A -85,B 0,C 180,E1 18039.104,E2 18039.104} C_VEL
LIN {X 0,Y 443.97,Z 882.665,A -85,B 0,C 180,E1 18041.766,E2 18041.766} C_VEL
LIN {X 0,Y 432.04,Z 919.567,A -85,B 0,C 180,E1 18045.034,E2 18045.034} C_VEL
LIN {X 0,Y 418.838,Z 955.352,A -85,B 0,C 180,E1 18049.365,E2 18049.365} C_VEL
LIN {X 0,Y 406.322,Z 986.998,A -85,B 0,C 180,E1 18054.642,E2 18054.642} C_VEL
LIN {X 0,Y 395.943,Z 1013.414,A -85,B 0,C 180,E1 18060.766,E2 18060.766} C_VEL
LIN {X 0,Y 388.554,Z 1034.275,A -85,B 0,C 180,E1 18067.651,E2 18067.651} C_VEL
LIN {X 0,Y 384.774,Z 1048.29,A -85,B 0,C 180,E1 18074.694,E2 18074.694} C_VEL
LIN {X 0,Y 383.231,Z 1055.84,A -85,B 0,C 180,E1 18081.35,E2 18081.35} C_VEL
LIN {X 0,Y 382.964,Z 1058.29,A -85,B 0,C 180,E1 18087.733,E2 18087.733} C_VEL
LIN {X 0,Y 383.236,Z 1057.012,A -85,B 0,C 180,E1 18092.267,E2 18092.267} C_VEL
LIN {X 0,Y 383.804,Z 1052.109,A -85,B 0,C 180,E1 18097.944,E2 18097.944} C_VEL
LIN {X 0,Y 386.2,Z 1040.883,A -85,B 0,C 180,E1 18104.778,E2 18104.778} C_VEL
LIN {X 0,Y 391.39,Z 1023.098,A -85,B 0,C 180,E1 18111.674,E2 18111.674} C_VEL
LIN {X 0,Y 399.292,Z 1000.822,A -85,B 0,C 180,E1 18117.706,E2 18117.706} C_VEL
LIN {X 0,Y 409.5,Z 973.726,A -85,B 0,C 180,E1 18123.083,E2 18123.083} C_VEL
LIN {X 0,Y 421.866,Z 940.203,A -85,B 0,C 180,E1 18127.964,E2 18127.964} C_VEL
LIN {X 0,Y 434.607,Z 902.155,A -85,B 0,C 180,E1 18131.994,E2 18131.994} C_VEL
LIN {X 0,Y 446.29,Z 860.864,A -85,B 0,C 180,E1 18135.151,E2 18135.151} C_VEL
LIN {X 0,Y 451.386,Z 838.321,A -85,B 0,C 180,E1 18136.484,E2 18136.484} C_VEL
LIN {X 0,Y 441.159,Z 806.432,A -85,B 0,C 180,E1 18140.54,E2 18140.54} C_VEL
LIN {X 0,Y 428.272,Z 778.098,A -85,B 0,C 180,E1 18144.741,E2 18144.741} C_VEL
LIN {X 0,Y 413.652,Z 752.854,A -85,B 0,C 180,E1 18149.369,E2 18149.369} C_VEL
LIN {X 0,Y 400.833,Z 734.548,A -85,B 0,C 180,E1 18153.698,E2 18153.698} C_VEL
LIN {X 0,Y 395.449,Z 727.461,A -85,B 0,C 180,E1 18155.744,E2 18155.744} C_VEL
LIN {X 0,Y 391.3,Z 721.546,A -85,B 0,C 180,E1 18157.512,E2 18157.512} C_VEL
LIN {X 0,Y 387.323,Z 716.068,A -85,B 0,C 180,E1 18159.379,E2 18159.379} C_VEL
LIN {X 0,Y 381.902,Z 709.574,A -85,B 0,C 180,E1 18162.259,E2 18162.259} C_VEL
LIN {X 0,Y 381.574,Z 707.31,A -85,B 0,C 180,E1 18162.779,E2 18162.779} C_VEL
LIN {X 0,Y 382.144,Z 707.31,A -85,B 0,C 180,E1 18168.56,E2 18168.56} C_VEL
LIN {X 0,Y 382.436,Z 707.31,A -85,B 0,C 180,E1 18175.45,E2 18175.45} C_VEL
LIN {X 0,Y 382.57,Z 707.31,A -85,B 0,C 180,E1 18182.266,E2 18182.266} C_VEL
LIN {X 0,Y 382.27,Z 707.31,A -85,B 0,C 180,E1 18189.12,E2 18189.12} C_VEL
LIN {X 0,Y 381.775,Z 708.18,A -85,B 0,C 180,E1 18195.168,E2 18195.168} C_VEL
LIN {X 0,Y 384.507,Z 713.459,A -85,B 0,C 180,E1 18196.819,E2 18196.819} C_VEL
LIN {X 0,Y 387.407,Z 715.926,A -85,B 0,C 180,E1 18198.231,E2 18198.231} C_VEL
LIN {X 0,Y 391.365,Z 721.533,A -85,B 0,C 180,E1 18200.095,E2 18200.095} C_VEL
LIN {X 0,Y 398.951,Z 731.904,A -85,B 0,C 180,E1 18203.187,E2 18203.187} C_VEL
LIN {X 0,Y 412.637,Z 750.952,A -85,B 0,C 180,E1 18207.804,E2 18207.804} C_VEL
LIN {X 0,Y 428.884,Z 777.324,A -85,B 0,C 180,E1 18212.6,E2 18212.6} C_VEL
LIN {X 0,Y 444.038,Z 809.072,A -85,B 0,C 180,E1 18217.102,E2 18217.102} C_VEL
LIN {X 0,Y 453.898,Z 837.297,A -85,B 0,C 180,E1 18220.489,E2 18220.489} C_VEL
LIN {X 0,Y 443.919,Z 880.92,A -85,B 0,C 180,E1 18222.868,E2 18222.868} C_VEL
LIN {X 0,Y 432.119,Z 921.786,A -85,B 0,C 180,E1 18226.017,E2 18226.017} C_VEL
LIN {X 0,Y 419.314,Z 959.996,A -85,B 0,C 180,E1 18230.096,E2 18230.096} C_VEL
LIN {X 0,Y 406.978,Z 993.964,A -85,B 0,C 180,E1 18235.088,E2 18235.088} C_VEL
LIN {X 0,Y 396.391,Z 1023.764,A -85,B 0,C 180,E1 18241.139,E2 18241.139} C_VEL
LIN {X 0,Y 388.913,Z 1046.788,A -85,B 0,C 180,E1 18247.671,E2 18247.671} C_VEL
LIN {X 0,Y 384.859,Z 1063.56,A -85,B 0,C 180,E1 18254.574,E2 18254.574} C_VEL
LIN {X 0,Y 383.359,Z 1073.624,A -85,B 0,C 180,E1 18261.172,E2 18261.172} C_VEL
LIN {X 0,Y 383.093,Z 1078.356,A -85,B 0,C 180,E1 18267.732,E2 18267.732} C_VEL
LIN {X 0,Y 383.204,Z 1078.425,A -85,B 0,C 180,E1 18272.265,E2 18272.265} C_VEL
LIN {X 0,Y 383.357,Z 1073.809,A -85,B 0,C 180,E1 18279.097,E2 18279.097} C_VEL
LIN {X 0,Y 384.936,Z 1064.503,A -85,B 0,C 180,E1 18285.441,E2 18285.441} C_VEL
LIN {X 0,Y 389.121,Z 1048.331,A -85,B 0,C 180,E1 18292.314,E2 18292.314} C_VEL
LIN {X 0,Y 396.733,Z 1025.8,A -85,B 0,C 180,E1 18298.909,E2 18298.909} C_VEL
LIN {X 0,Y 407.034,Z 998.456,A -85,B 0,C 180,E1 18304.675,E2 18304.675} C_VEL
LIN {X 0,Y 419.176,Z 966.787,A -85,B 0,C 180,E1 18309.58,E2 18309.58} C_VEL
LIN {X 0,Y 432.108,Z 930.978,A -85,B 0,C 180,E1 18313.664,E2 18313.664} C_VEL
LIN {X 0,Y 434.024,Z 925.236,A -85,B 0,C 180,E1 18314.208,E2 18314.208} C_VEL
LIN {X 0,Y 435.463,Z 912.16,A -85,B 0,C 180,E1 18315.745,E2 18315.745} C_VEL
LIN {X 0,Y 436.537,Z 900.432,A -85,B 0,C 180,E1 18317.033,E2 18317.033} C_VEL
LIN {X 0,Y 437.069,Z 898.583,A -85,B 0,C 180,E1 18317.176,E2 18317.176} C_VEL
LIN {X 0,Y 448.356,Z 858.202,A -85,B 0,C 180,E1 18319.738,E2 18319.738} C_VEL
LIN {X 0,Y 451.986,Z 843.433,A -85,B 0,C 180,E1 18320.454,E2 18320.454} C_VEL
LIN {X 0,Y 442.735,Z 815.835,A -85,B 0,C 180,E1 18324.12,E2 18324.12} C_VEL
LIN {X 0,Y 429.535,Z 787.822,A -85,B 0,C 180,E1 18328.642,E2 18328.642} C_VEL
LIN {X 0,Y 415.222,Z 763.142,A -85,B 0,C 180,E1 18333.74,E2 18333.74} C_VEL
LIN {X 0,Y 401.852,Z 743.819,A -85,B 0,C 180,E1 18339.229,E2 18339.229} C_VEL
LIN {X 0,Y 395.7,Z 736.14,A -85,B 0,C 180,E1 18342.308,E2 18342.308} C_VEL
LIN {X 0,Y 391.373,Z 729.771,A -85,B 0,C 180,E1 18344.997,E2 18344.997} C_VEL
LIN {X 0,Y 387.3,Z 724.158,A -85,B 0,C 180,E1 18348.136,E2 18348.136} C_VEL
LIN {X 0,Y 385.799,Z 722.349,A -85,B 0,C 180,E1 18349.537,E2 18349.537} C_VEL
LIN {X 0,Y 381.428,Z 715.38,A -85,B 0,C 180,E1 18357.229,E2 18357.229} C_VEL
LIN {X 0,Y 381.395,Z 715.994,A -85,B 0,C 180,E1 18361.285,E2 18361.285} C_VEL
LIN {X 0,Y 387.187,Z 723.796,A -85,B 0,C 180,E1 18370.077,E2 18370.077} C_VEL
LIN {X 0,Y 390.847,Z 729.352,A -85,B 0,C 180,E1 18372.997,E2 18372.997} C_VEL
LIN {X 0,Y 392.877,Z 731.674,A -85,B 0,C 180,E1 18374.31,E2 18374.31} C_VEL
LIN {X 0,Y 398.85,Z 740.075,A -85,B 0,C 180,E1 18377.699,E2 18377.699} C_VEL
LIN {X 0,Y 407.645,Z 752.199,A -85,B 0,C 180,E1 18381.745,E2 18381.745} C_VEL
LIN {X 0,Y 421.733,Z 774.941,A -85,B 0,C 180,E1 18387.343,E2 18387.343} C_VEL
LIN {X 0,Y 435.305,Z 802.391,A -85,B 0,C 180,E1 18392.396,E2 18392.396} C_VEL
LIN {X 0,Y 446.054,Z 831.504,A -85,B 0,C 180,E1 18396.787,E2 18396.787} C_VEL
LIN {X 0,Y 449.234,Z 844.626,A -85,B 0,C 180,E1 18398.509,E2 18398.509} C_VEL
LIN {X 0,Y 436.834,Z 888.399,A -85,B 0,C 180,E1 18401.417,E2 18401.417} C_VEL
LIN {X 0,Y 423.575,Z 927.066,A -85,B 0,C 180,E1 18405.066,E2 18405.066} C_VEL
LIN {X 0,Y 410.46,Z 960.773,A -85,B 0,C 180,E1 18409.427,E2 18409.427} C_VEL
LIN {X 0,Y 398.436,Z 989.93,A -85,B 0,C 180,E1 18414.55,E2 18414.55} C_VEL
LIN {X 0,Y 387.99,Z 1015.609,A -85,B 0,C 180,E1 18420.778,E2 18420.778} C_VEL
LIN {X 0,Y 381.024,Z 1034.425,A -85,B 0,C 180,E1 18427.185,E2 18427.185} C_VEL
LIN {X 0,Y 377.255,Z 1047.338,A -85,B 0,C 180,E1 18433.67,E2 18433.67} C_VEL
LIN {X 0,Y 375.601,Z 1054.737,A -85,B 0,C 180,E1 18439.541,E2 18439.541} C_VEL
LIN {X 0,Y 375.028,Z 1058.177,A -85,B 0,C 180,E1 18445.366,E2 18445.366} C_VEL
LIN {X 0,Y 375.365,Z 1058.162,A -85,B 0,C 180,E1 18450.001,E2 18450.001} C_VEL
LIN {X 0,Y 375.714,Z 1053.575,A -85,B 0,C 180,E1 18456.951,E2 18456.951} C_VEL
LIN {X 0,Y 377.601,Z 1044.517,A -85,B 0,C 180,E1 18463.343,E2 18463.343} C_VEL
LIN {X 0,Y 382.21,Z 1028.728,A -85,B 0,C 180,E1 18470.3,E2 18470.3} C_VEL
LIN {X 0,Y 390.211,Z 1006.382,A -85,B 0,C 180,E1 18476.994,E2 18476.994} C_VEL
LIN {X 0,Y 401.652,Z 977.2,A -85,B 0,C 180,E1 18483.168,E2 18483.168} C_VEL
LIN {X 0,Y 414.87,Z 942.661,A -85,B 0,C 180,E1 18488.387,E2 18488.387} C_VEL
LIN {X 0,Y 428.312,Z 903.963,A -85,B 0,C 180,E1 18492.584,E2 18492.584} C_VEL
LIN {X 0,Y 440.739,Z 861.478,A -85,B 0,C 180,E1 18495.87,E2 18495.87} C_VEL
LIN {X 0,Y 445.378,Z 841.149,A -85,B 0,C 180,E1 18497.113,E2 18497.113} C_VEL
LIN {X 0,Y 435.628,Z 809.93,A -85,B 0,C 180,E1 18501.229,E2 18501.229} C_VEL
LIN {X 0,Y 423.277,Z 781.882,A -85,B 0,C 180,E1 18505.539,E2 18505.539} C_VEL
LIN {X 0,Y 407.953,Z 755.111,A -85,B 0,C 180,E1 18510.701,E2 18510.701} C_VEL
LIN {X 0,Y 394.182,Z 735.467,A -85,B 0,C 180,E1 18515.812,E2 18515.812} C_VEL
LIN {X 0,Y 388.822,Z 728.455,A -85,B 0,C 180,E1 18518.114,E2 18518.114} C_VEL
LIN {X 0,Y 383.917,Z 721.777,A -85,B 0,C 180,E1 18520.542,E2 18520.542} C_VEL
LIN {X 0,Y 379.995,Z 716.405,A -85,B 0,C 180,E1 18522.792,E2 18522.792} C_VEL
LIN {X 0,Y 378.528,Z 714.528,A -85,B 0,C 180,E1 18523.721,E2 18523.721} C_VEL
LIN {X 0,Y 374.447,Z 709.771,A -85,B 0,C 180,E1 18526.674,E2 18526.674} C_VEL
LIN {X 0,Y 374.109,Z 707.31,A -85,B 0,C 180,E1 18527.487,E2 18527.487} C_VEL
LIN {X 0,Y 374.535,Z 707.31,A -85,B 0,C 180,E1 18533.024,E2 18533.024} C_VEL
LIN {X 0,Y 374.714,Z 707.31,A -85,B 0,C 180,E1 18539.996,E2 18539.996} C_VEL
LIN {X 0,Y 374.418,Z 707.31,A -85,B 0,C 180,E1 18546.97,E2 18546.97} C_VEL
LIN {X 0,Y 374.206,Z 707.956,A -85,B 0,C 180,E1 18550.569,E2 18550.569} C_VEL
LIN {X 0,Y 376.846,Z 713.387,A -85,B 0,C 180,E1 18552.79,E2 18552.79} C_VEL
LIN {X 0,Y 380.046,Z 716.088,A -85,B 0,C 180,E1 18554.795,E2 18554.795} C_VEL
LIN {X 0,Y 383.862,Z 721.701,A -85,B 0,C 180,E1 18557.011,E2 18557.011} C_VEL
LIN {X 0,Y 385.873,Z 724.237,A -85,B 0,C 180,E1 18558.04,E2 18558.04} C_VEL
LIN {X 0,Y 391.793,Z 732.31,A -85,B 0,C 180,E1 18560.778,E2 18560.778} C_VEL
LIN {X 0,Y 401.303,Z 745.199,A -85,B 0,C 180,E1 18564.463,E2 18564.463} C_VEL
LIN {X 0,Y 416.1,Z 767.521,A -85,B 0,C 180,E1 18569.37,E2 18569.37} C_VEL
LIN {X 0,Y 431.65,Z 796.46,A -85,B 0,C 180,E1 18574.17,E2 18574.17} C_VEL
LIN {X 0,Y 444.19,Z 827.856,A -85,B 0,C 180,E1 18578.371,E2 18578.371} C_VEL
LIN {X 0,Y 447.793,Z 842.158,A -85,B 0,C 180,E1 18579.981,E2 18579.981} C_VEL
LIN {X 0,Y 437.193,Z 885.036,A -85,B 0,C 180,E1 18582.399,E2 18582.399} C_VEL
LIN {X 0,Y 425.295,Z 924.395,A -85,B 0,C 180,E1 18585.542,E2 18585.542} C_VEL
LIN {X 0,Y 412.343,Z 961.609,A -85,B 0,C 180,E1 18589.628,E2 18589.628} C_VEL
LIN {X 0,Y 399.622,Z 995.441,A -85,B 0,C 180,E1 18594.736,E2 18594.736} C_VEL
LIN {X 0,Y 388.801,Z 1024.667,A -85,B 0,C 180,E1 18600.855,E2 18600.855} C_VEL
LIN {X 0,Y 381.4,Z 1046.515,A -85,B 0,C 180,E1 18607.207,E2 18607.207} C_VEL
LIN {X 0,Y 377.298,Z 1062.156,A -85,B 0,C 180,E1 18613.67,E2 18613.67} C_VEL
LIN {X 0,Y 375.676,Z 1071.729,A -85,B 0,C 180,E1 18619.541,E2 18619.541} C_VEL
LIN {X 0,Y 375.143,Z 1077.095,A -85,B 0,C 180,E1 18625.365,E2 18625.365} C_VEL
LIN {X 0,Y 375.353,Z 1078.499,A -85,B 0,C 180,E1 18629.999,E2 18629.999} C_VEL
LIN {X 0,Y 375.315,Z 1075.778,A -85,B 0,C 180,E1 18636.956,E2 18636.956} C_VEL
LIN {X 0,Y 376.109,Z 1069.211,A -85,B 0,C 180,E1 18642.802,E2 18642.802} C_VEL
LIN {X 0,Y 379.423,Z 1055.348,A -85,B 0,C 180,E1 18649.989,E2 18649.989} C_VEL
LIN {X 0,Y 385.124,Z 1037.415,A -85,B 0,C 180,E1 18656.273,E2 18656.273} C_VEL
LIN {X 0,Y 394.616,Z 1012.625,A -85,B 0,C 180,E1 18662.521,E2 18662.521} C_VEL
LIN {X 0,Y 407.179,Z 981.515,A -85,B 0,C 180,E1 18668.168,E2 18668.168} C_VEL
LIN {X 0,Y 420.85,Z 946.258,A -85,B 0,C 180,E1 18672.807,E2 18672.807} C_VEL
LIN {X 0,Y 434.958,Z 905.458,A -85,B 0,C 180,E1 18676.658,E2 18676.658} C_VEL
LIN {X 0,Y 437.069,Z 898.583,A -85,B 0,C 180,E1 18677.176,E2 18677.176} C_VEL
LIN {X 0,Y 437.14,Z 889.705,A -85,B 0,C 180,E1 18678.207,E2 18678.207} C_VEL
LIN {X 0,Y 437.081,Z 880.685,A -85,B 0,C 180,E1 18679.212,E2 18679.212} C_VEL
LIN {X 0,Y 446.074,Z 844.945,A -85,B 0,C 180,E1 18681.272,E2 18681.272} C_VEL
LIN {X 0,Y 435.501,Z 814.666,A -85,B 0,C 180,E1 18685.572,E2 18685.572} C_VEL
LIN {X 0,Y 421.782,Z 786.054,A -85,B 0,C 180,E1 18690.578,E2 18690.578} C_VEL
LIN {X 0,Y 408.11,Z 763.363,A -85,B 0,C 180,E1 18695.897,E2 18695.897} C_VEL
LIN {X 0,Y 398.664,Z 749.922,A -85,B 0,C 180,E1 18700.144,E2 18700.144} C_VEL
LIN {X 0,Y 393.904,Z 743.354,A -85,B 0,C 180,E1 18702.73,E2 18702.73} C_VEL
LIN {X 0,Y 389.791,Z 737.299,A -85,B 0,C 180,E1 18705.367,E2 18705.367} C_VEL
LIN {X 0,Y 385.745,Z 731.049,A -85,B 0,C 180,E1 18708.676,E2 18708.676} C_VEL
LIN {X 0,Y 380.402,Z 722.941,A -85,B 0,C 180,E1 18717.721,E2 18717.721} C_VEL
LIN {X 0,Y 380.411,Z 724.004,A -85,B 0,C 180,E1 18721.288,E2 18721.288} C_VEL
LIN {X 0,Y 385.892,Z 731.569,A -85,B 0,C 180,E1 18729.826,E2 18729.826} C_VEL
LIN {X 0,Y 389.901,Z 737.256,A -85,B 0,C 180,E1 18733.029,E2 18733.029} C_VEL
LIN {X 0,Y 397.082,Z 747.576,A -85,B 0,C 180,E1 18737.433,E2 18737.433} C_VEL
LIN {X 0,Y 405.808,Z 760.44,A -85,B 0,C 180,E1 18741.683,E2 18741.683} C_VEL
LIN {X 0,Y 418.357,Z 781.433,A -85,B 0,C 180,E1 18746.926,E2 18746.926} C_VEL
LIN {X 0,Y 431.328,Z 809.029,A -85,B 0,C 180,E1 18752.128,E2 18752.128} C_VEL
LIN {X 0,Y 441.361,Z 838.37,A -85,B 0,C 180,E1 18756.635,E2 18756.635} C_VEL
LIN {X 0,Y 443.584,Z 846.974,A -85,B 0,C 180,E1 18757.819,E2 18757.819} C_VEL
LIN {X 0,Y 430.772,Z 890.809,A -85,B 0,C 180,E1 18760.805,E2 18760.805} C_VEL
LIN {X 0,Y 416.194,Z 931.49,A -85,B 0,C 180,E1 18764.766,E2 18764.766} C_VEL
LIN {X 0,Y 401.799,Z 966.969,A -85,B 0,C 180,E1 18769.624,E2 18769.624} C_VEL
LIN {X 0,Y 388.641,Z 997.359,A -85,B 0,C 180,E1 18775.427,E2 18775.427} C_VEL
LIN {X 0,Y 378.204,Z 1022.233,A -85,B 0,C 180,E1 18782.161,E2 18782.161} C_VEL
LIN {X 0,Y 371.695,Z 1040.253,A -85,B 0,C 180,E1 18789.26,E2 18789.26} C_VEL
LIN {X 0,Y 368.622,Z 1050.949,A -85,B 0,C 180,E1 18795.721,E2 18795.721} C_VEL
LIN {X 0,Y 367.322,Z 1056.931,A -85,B 0,C 180,E1 18801.968,E2 18801.968} C_VEL
LIN {X 0,Y 367.155,Z 1058.711,A -85,B 0,C 180,E1 18807.636,E2 18807.636} C_VEL
LIN {X 0,Y 367.44,Z 1057.456,A -85,B 0,C 180,E1 18812.365,E2 18812.365} C_VEL
LIN {X 0,Y 368.205,Z 1051.74,A -85,B 0,C 180,E1 18818.953,E2 18818.953} C_VEL
LIN {X 0,Y 371.067,Z 1040.276,A -85,B 0,C 180,E1 18825.991,E2 18825.991} C_VEL
LIN {X 0,Y 377.235,Z 1021.911,A -85,B 0,C 180,E1 18833.176,E2 18833.176} C_VEL
LIN {X 0,Y 387.072,Z 996.705,A -85,B 0,C 180,E1 18839.946,E2 18839.946} C_VEL
LIN {X 0,Y 399.575,Z 966.106,A -85,B 0,C 180,E1 18845.757,E2 18845.757} C_VEL
LIN {X 0,Y 413.323,Z 930.596,A -85,B 0,C 180,E1 18850.602,E2 18850.602} C_VEL
LIN {X 0,Y 426.98,Z 890.662,A -85,B 0,C 180,E1 18854.504,E2 18854.504} C_VEL
LIN {X 0,Y 438.789,Z 848.655,A -85,B 0,C 180,E1 18857.416,E2 18857.416} C_VEL
LIN {X 0,Y 439.18,Z 842.925,A -85,B 0,C 180,E1 18857.891,E2 18857.891} C_VEL
LIN {X 0,Y 429.71,Z 812.042,A -85,B 0,C 180,E1 18862.122,E2 18862.122} C_VEL
LIN {X 0,Y 416.941,Z 783.117,A -85,B 0,C 180,E1 18866.827,E2 18866.827} C_VEL
LIN {X 0,Y 403.366,Z 759.629,A -85,B 0,C 180,E1 18871.682,E2 18871.682} C_VEL
LIN {X 0,Y 391.832,Z 742.414,A -85,B 0,C 180,E1 18876.264,E2 18876.264} C_VEL
LIN {X 0,Y 385.975,Z 734.734,A -85,B 0,C 180,E1 18878.927,E2 18878.927} C_VEL
LIN {X 0,Y 382.175,Z 729.222,A -85,B 0,C 180,E1 18880.901,E2 18880.901} C_VEL
LIN {X 0,Y 378.129,Z 723.195,A -85,B 0,C 180,E1 18883.33,E2 18883.33} C_VEL
LIN {X 0,Y 373.023,Z 717.224,A -85,B 0,C 180,E1 18887.028,E2 18887.028} C_VEL
LIN {X 0,Y 372.464,Z 715.033,A -85,B 0,C 180,E1 18887.662,E2 18887.662} C_VEL
LIN {X 0,Y 366.534,Z 707.565,A -85,B 0,C 180,E1 18897.182,E2 18897.182} C_VEL
LIN {X 0,Y 366.766,Z 708.138,A -85,B 0,C 180,E1 18901.623,E2 18901.623} C_VEL
LIN {X 0,Y 371.172,Z 714.563,A -85,B 0,C 180,E1 18908.802,E2 18908.802} C_VEL
LIN {X 0,Y 372.84,Z 716.106,A -85,B 0,C 180,E1 18910.312,E2 18910.312} C_VEL
LIN {X 0,Y 376.182,Z 721.537,A -85,B 0,C 180,E1 18913.013,E2 18913.013} C_VEL
LIN {X 0,Y 378.492,Z 723.866,A -85,B 0,C 180,E1 18914.496,E2 18914.496} C_VEL
LIN {X 0,Y 382.927,Z 729.661,A -85,B 0,C 180,E1 18917.053,E2 18917.053} C_VEL
LIN {X 0,Y 394.297,Z 745.554,A -85,B 0,C 180,E1 18922.268,E2 18922.268} C_VEL
LIN {X 0,Y 407.995,Z 766.003,A -85,B 0,C 180,E1 18927.303,E2 18927.303} C_VEL
LIN {X 0,Y 422.779,Z 792.529,A -85,B 0,C 180,E1 18932.215,E2 18932.215} C_VEL
LIN {X 0,Y 435.889,Z 823.552,A -85,B 0,C 180,E1 18936.735,E2 18936.735} C_VEL
LIN {X 0,Y 442.204,Z 844.041,A -85,B 0,C 180,E1 18939.301,E2 18939.301} C_VEL
LIN {X 0,Y 430.679,Z 888.496,A -85,B 0,C 180,E1 18941.872,E2 18941.872} C_VEL
LIN {X 0,Y 417.813,Z 929.045,A -85,B 0,C 180,E1 18945.251,E2 18945.251} C_VEL
LIN {X 0,Y 405.407,Z 963.209,A -85,B 0,C 180,E1 18949.144,E2 18949.144} C_VEL
LIN {X 0,Y 392.491,Z 996.275,A -85,B 0,C 180,E1 18954.261,E2 18954.261} C_VEL
LIN {X 0,Y 381.662,Z 1024.335,A -85,B 0,C 180,E1 18960.244,E2 18960.244} C_VEL
LIN {X 0,Y 373.881,Z 1046.24,A -85,B 0,C 180,E1 18966.721,E2 18966.721} C_VEL
LIN {X 0,Y 369.308,Z 1063.003,A -85,B 0,C 180,E1 18973.881,E2 18973.881} C_VEL
LIN {X 0,Y 367.619,Z 1072.867,A -85,B 0,C 180,E1 18980.508,E2 18980.508} C_VEL
LIN {X 0,Y 367.241,Z 1076.876,A -85,B 0,C 180,E1 18985.265,E2 18985.265} C_VEL
LIN {X 0,Y 367.452,Z 1078.286,A -85,B 0,C 180,E1 18989.999,E2 18989.999} C_VEL
LIN {X 0,Y 367.413,Z 1075.579,A -85,B 0,C 180,E1 18997.107,E2 18997.107} C_VEL
LIN {X 0,Y 368.299,Z 1069.021,A -85,B 0,C 180,E1 19003.078,E2 19003.078} C_VEL
LIN {X 0,Y 371.771,Z 1055.268,A -85,B 0,C 180,E1 19010.375,E2 19010.375} C_VEL
LIN {X 0,Y 377.843,Z 1037.262,A -85,B 0,C 180,E1 19016.819,E2 19016.819} C_VEL
LIN {X 0,Y 387.806,Z 1012.496,A -85,B 0,C 180,E1 19023.165,E2 19023.165} C_VEL
LIN {X 0,Y 400.519,Z 982.187,A -85,B 0,C 180,E1 19028.768,E2 19028.768} C_VEL
LIN {X 0,Y 415.214,Z 945.485,A -85,B 0,C 180,E1 19033.643,E2 19033.643} C_VEL
LIN {X 0,Y 429.504,Z 905.45,A -85,B 0,C 180,E1 19037.435,E2 19037.435} C_VEL
LIN {X 0,Y 437.081,Z 880.685,A -85,B 0,C 180,E1 19039.212,E2 19039.212} C_VEL
LIN {X 0,Y 438.779,Z 866.169,A -85,B 0,C 180,E1 19040.474,E2 19040.474} C_VEL
LIN {X 0,Y 440.119,Z 851.31,A -85,B 0,C 180,E1 19041.672,E2 19041.672} C_VEL
LIN {X 0,Y 439.685,Z 845.5,A -85,B 0,C 180,E1 19042.288,E2 19042.288} C_VEL
LIN {X 0,Y 429.054,Z 815.352,A -85,B 0,C 180,E1 19046.812,E2 19046.812} C_VEL
LIN {X 0,Y 415.682,Z 787.53,A -85,B 0,C 180,E1 19052.039,E2 19052.039} C_VEL
LIN {X 0,Y 403.691,Z 767.569,A -85,B 0,C 180,E1 19057.083,E2 19057.083} C_VEL
LIN {X 0,Y 396.097,Z 756.398,A -85,B 0,C 180,E1 19060.81,E2 19060.81} C_VEL
LIN {X 0,Y 391.875,Z 750.439,A -85,B 0,C 180,E1 19063.217,E2 19063.217} C_VEL
LIN {X 0,Y 388.204,Z 744.799,A -85,B 0,C 180,E1 19065.739,E2 19065.739} C_VEL
LIN {X 0,Y 383.606,Z 737.901,A -85,B 0,C 180,E1 19069.765,E2 19069.765} C_VEL
LIN {X 0,Y 379.439,Z 730.788,A -85,B 0,C 180,E1 19077.715,E2 19077.715} C_VEL
LIN {X 0,Y 379.421,Z 731.793,A -85,B 0,C 180,E1 19081.148,E2 19081.148} C_VEL
LIN {X 0,Y 384.674,Z 739.452,A -85,B 0,C 180,E1 19089.642,E2 19089.642} C_VEL
LIN {X 0,Y 389.953,Z 747.381,A -85,B 0,C 180,E1 19093.917,E2 19093.917} C_VEL
LIN {X 0,Y 396.042,Z 756.331,A -85,B 0,C 180,E1 19097.611,E2 19097.611} C_VEL
LIN {X 0,Y 406.266,Z 772.259,A -85,B 0,C 180,E1 19102.699,E2 19102.699} C_VEL
LIN {X 0,Y 418.385,Z 795.084,A -85,B 0,C 180,E1 19108.021,E2 19108.021} C_VEL
LIN {X 0,Y 429.665,Z 821.911,A -85,B 0,C 180,E1 19112.918,E2 19112.918} C_VEL
LIN {X 0,Y 437.563,Z 849.06,A -85,B 0,C 180,E1 19117.029,E2 19117.029} C_VEL
LIN {X 0,Y 435.507,Z 859.052,A -85,B 0,C 180,E1 19117.746,E2 19117.746} C_VEL
LIN {X 0,Y 422.739,Z 898.804,A -85,B 0,C 180,E1 19120.673,E2 19120.673} C_VEL
LIN {X 0,Y 408.775,Z 935.731,A -85,B 0,C 180,E1 19124.47,E2 19124.47} C_VEL
LIN {X 0,Y 394.601,Z 969.305,A -85,B 0,C 180,E1 19129.244,E2 19129.244} C_VEL
LIN {X 0,Y 382.143,Z 996.986,A -85,B 0,C 180,E1 19134.619,E2 19134.619} C_VEL
LIN {X 0,Y 371.434,Z 1021.334,A -85,B 0,C 180,E1 19141.238,E2 19141.238} C_VEL
LIN {X 0,Y 364.138,Z 1040.207,A -85,B 0,C 180,E1 19148.709,E2 19148.709} C_VEL
LIN {X 0,Y 360.824,Z 1051.13,A -85,B 0,C 180,E1 19155.406,E2 19155.406} C_VEL
LIN {X 0,Y 359.695,Z 1056.092,A -85,B 0,C 180,E1 19160.299,E2 19160.299} C_VEL
LIN {X 0,Y 359.278,Z 1058.919,A -85,B 0,C 180,E1 19167.584,E2 19167.584} C_VEL
LIN {X 0,Y 359.554,Z 1057.678,A -85,B 0,C 180,E1 19172.417,E2 19172.417} C_VEL
LIN {X 0,Y 360.28,Z 1052.431,A -85,B 0,C 180,E1 19178.797,E2 19178.797} C_VEL
LIN {X 0,Y 362.915,Z 1042.135,A -85,B 0,C 180,E1 19185.492,E2 19185.492} C_VEL
LIN {X 0,Y 368.439,Z 1025.731,A -85,B 0,C 180,E1 19192.436,E2 19192.436} C_VEL
LIN {X 0,Y 377.102,Z 1004.137,A -85,B 0,C 180,E1 19198.832,E2 19198.832} C_VEL
LIN {X 0,Y 388.68,Z 976.941,A -85,B 0,C 180,E1 19204.638,E2 19204.638} C_VEL
LIN {X 0,Y 402.86,Z 942.405,A -85,B 0,C 180,E1 19209.929,E2 19209.929} C_VEL
LIN {X 0,Y 417.096,Z 903.925,A -85,B 0,C 180,E1 19214.139,E2 19214.139} C_VEL
LIN {X 0,Y 429.88,Z 862.462,A -85,B 0,C 180,E1 19217.383,E2 19217.383} C_VEL
LIN {X 0,Y 433.57,Z 847.102,A -85,B 0,C 180,E1 19218.384,E2 19218.384} C_VEL
LIN {X 0,Y 424.38,Z 815.809,A -85,B 0,C 180,E1 19222.818,E2 19222.818} C_VEL
LIN {X 0,Y 411.929,Z 786.988,A -85,B 0,C 180,E1 19227.695,E2 19227.695} C_VEL
LIN {X 0,Y 398.272,Z 762.588,A -85,B 0,C 180,E1 19232.972,E2 19232.972} C_VEL
LIN {X 0,Y 385.639,Z 743.639,A -85,B 0,C 180,E1 19238.53,E2 19238.53} C_VEL
LIN {X 0,Y 379.557,Z 735.857,A -85,B 0,C 180,E1 19241.746,E2 19241.746} C_VEL
LIN {X 0,Y 375.524,Z 729.77,A -85,B 0,C 180,E1 19244.339,E2 19244.339} C_VEL
LIN {X 0,Y 371.393,Z 723.954,A -85,B 0,C 180,E1 19247.626,E2 19247.626} C_VEL
LIN {X 0,Y 369.295,Z 722.003,A -85,B 0,C 180,E1 19249.654,E2 19249.654} C_VEL
LIN {X 0,Y 365.537,Z 715.134,A -85,B 0,C 180,E1 19257.62,E2 19257.62} C_VEL
LIN {X 0,Y 365.822,Z 716.213,A -85,B 0,C 180,E1 19261.776,E2 19261.776} C_VEL
LIN {X 0,Y 369.91,Z 722.287,A -85,B 0,C 180,E1 19268.536,E2 19268.536} C_VEL
LIN {X 0,Y 371.583,Z 724.182,A -85,B 0,C 180,E1 19270.125,E2 19270.125} C_VEL
LIN {X 0,Y 375.529,Z 729.644,A -85,B 0,C 180,E1 19273.237,E2 19273.237} C_VEL
LIN {X 0,Y 377.753,Z 733.204,A -85,B 0,C 180,E1 19274.739,E2 19274.739} C_VEL
LIN {X 0,Y 382.791,Z 739.922,A -85,B 0,C 180,E1 19277.587,E2 19277.587} C_VEL
LIN {X 0,Y 391.506,Z 751.784,A -85,B 0,C 180,E1 19281.653,E2 19281.653} C_VEL
LIN {X 0,Y 405.341,Z 773.273,A -85,B 0,C 180,E1 19287.026,E2 19287.026} C_VEL
LIN {X 0,Y 419.529,Z 800.132,A -85,B 0,C 180,E1 19292.037,E2 19292.037} C_VEL
LIN {X 0,Y 431.507,Z 830.183,A -85,B 0,C 180,E1 19296.48,E2 19296.48} C_VEL
LIN {X 0,Y 436.109,Z 848.118,A -85,B 0,C 180,E1 19298.711,E2 19298.711} C_VEL
LIN {X 0,Y 424.022,Z 892.426,A -85,B 0,C 180,E1 19301.364,E2 19301.364} C_VEL
LIN {X 0,Y 410.158,Z 934.179,A -85,B 0,C 180,E1 19305.002,E2 19305.002} C_VEL
LIN {X 0,Y 395.487,Z 972.478,A -85,B 0,C 180,E1 19309.708,E2 19309.708} C_VEL
LIN {X 0,Y 382.305,Z 1004.857,A -85,B 0,C 180,E1 19315.262,E2 19315.262} C_VEL
LIN {X 0,Y 371.643,Z 1031.823,A -85,B 0,C 180,E1 19321.715,E2 19321.715} C_VEL
LIN {X 0,Y 364.331,Z 1052.358,A -85,B 0,C 180,E1 19328.66,E2 19328.66} C_VEL
LIN {X 0,Y 360.877,Z 1065.997,A -85,B 0,C 180,E1 19335.406,E2 19335.406} C_VEL
LIN {X 0,Y 359.656,Z 1073.828,A -85,B 0,C 180,E1 19341.472,E2 19341.472} C_VEL
LIN {X 0,Y 359.393,Z 1077.708,A -85,B 0,C 180,E1 19347.582,E2 19347.582} C_VEL
LIN {X 0,Y 359.49,Z 1077.799,A -85,B 0,C 180,E1 19352.415,E2 19352.415} C_VEL
LIN {X 0,Y 359.708,Z 1073.226,A -85,B 0,C 180,E1 19359.7,E2 19359.7} C_VEL
LIN {X 0,Y 361.437,Z 1064.705,A -85,B 0,C 180,E1 19366.012,E2 19366.012} C_VEL
LIN {X 0,Y 366.084,Z 1049.385,A -85,B 0,C 180,E1 19373.156,E2 19373.156} C_VEL
LIN {X 0,Y 374.22,Z 1028.346,A -85,B 0,C 180,E1 19379.915,E2 19379.915} C_VEL
LIN {X 0,Y 385.11,Z 1002.875,A -85,B 0,C 180,E1 19385.825,E2 19385.825} C_VEL
LIN {X 0,Y 399.138,Z 970.377,A -85,B 0,C 180,E1 19391.274,E2 19391.274} C_VEL
LIN {X 0,Y 414.402,Z 932.411,A -85,B 0,C 180,E1 19395.815,E2 19395.815} C_VEL
LIN {X 0,Y 428.933,Z 890.665,A -85,B 0,C 180,E1 19399.342,E2 19399.342} C_VEL
LIN {X 0,Y 440.119,Z 851.31,A -85,B 0,C 180,E1 19401.672,E2 19401.672} C_VEL
LIN {X 0,Y 439.625,Z 844.958,A -85,B 0,C 180,E1 19402.344,E2 19402.344} C_VEL
LIN {X 0,Y 429.034,Z 832.724,A -85,B 0,C 180,E1 19405.353,E2 19405.353} C_VEL
LIN {X 0,Y 417.28,Z 803.995,A -85,B 0,C 180,E1 19410.368,E2 19410.368} C_VEL
LIN {X 0,Y 405.39,Z 781.612,A -85,B 0,C 180,E1 19415.488,E2 19415.488} C_VEL
LIN {X 0,Y 395.298,Z 765.25,A -85,B 0,C 180,E1 19420.478,E2 19420.478} C_VEL
LIN {X 0,Y 386.889,Z 752.538,A -85,B 0,C 180,E1 19425.834,E2 19425.834} C_VEL
LIN {X 0,Y 382.305,Z 745.621,A -85,B 0,C 180,E1 19430.018,E2 19430.018} C_VEL
LIN {X 0,Y 378.362,Z 738.604,A -85,B 0,C 180,E1 19438.857,E2 19438.857} C_VEL
LIN {X 0,Y 378.503,Z 740.325,A -85,B 0,C 180,E1 19441.653,E2 19441.653} C_VEL
LIN {X 0,Y 383.226,Z 747.16,A -85,B 0,C 180,E1 19449.392,E2 19449.392} C_VEL
LIN {X 0,Y 388.378,Z 755.057,A -85,B 0,C 180,E1 19453.687,E2 19453.687} C_VEL
LIN {X 0,Y 396.019,Z 766.493,A -85,B 0,C 180,E1 19458.479,E2 19458.479} C_VEL
LIN {X 0,Y 407.639,Z 787.019,A -85,B 0,C 180,E1 19464.36,E2 19464.36} C_VEL
LIN {X 0,Y 418.487,Z 810.207,A -85,B 0,C 180,E1 19469.388,E2 19469.388} C_VEL
LIN {X 0,Y 428.2,Z 837.878,A -85,B 0,C 180,E1 19474.185,E2 19474.185} C_VEL
LIN {X 0,Y 431.953,Z 853.965,A -85,B 0,C 180,E1 19476.586,E2 19476.586} C_VEL
LIN {X 0,Y 418.842,Z 895.093,A -85,B 0,C 180,E1 19479.512,E2 19479.512} C_VEL
LIN {X 0,Y 404.022,Z 933.672,A -85,B 0,C 180,E1 19483.39,E2 19483.39} C_VEL
LIN {X 0,Y 389.203,Z 967.784,A -85,B 0,C 180,E1 19488.181,E2 19488.181} C_VEL
LIN {X 0,Y 375.358,Z 997.397,A -85,B 0,C 180,E1 19493.964,E2 19493.964} C_VEL
LIN {X 0,Y 363.699,Z 1022.784,A -85,B 0,C 180,E1 19501.052,E2 19501.052} C_VEL
LIN {X 0,Y 356.274,Z 1041.259,A -85,B 0,C 180,E1 19508.68,E2 19508.68} C_VEL
LIN {X 0,Y 352.674,Z 1052.847,A -85,B 0,C 180,E1 19516.331,E2 19516.331} C_VEL
LIN {X 0,Y 351.473,Z 1057.868,A -85,B 0,C 180,E1 19522.624,E2 19522.624} C_VEL
LIN {X 0,Y 351.657,Z 1058.805,A -85,B 0,C 180,E1 19530.001,E2 19530.001} C_VEL
LIN {X 0,Y 352.122,Z 1054.287,A -85,B 0,C 180,E1 19537.419,E2 19537.419} C_VEL
LIN {X 0,Y 354.341,Z 1045.303,A -85,B 0,C 180,E1 19544.237,E2 19544.237} C_VEL
LIN {X 0,Y 359.708,Z 1029.566,A -85,B 0,C 180,E1 19551.632,E2 19551.632} C_VEL
LIN {X 0,Y 369.124,Z 1006.767,A -85,B 0,C 180,E1 19558.842,E2 19558.842} C_VEL
LIN {X 0,Y 381.761,Z 978.069,A -85,B 0,C 180,E1 19565.176,E2 19565.176} C_VEL
LIN {X 0,Y 396.369,Z 943.8,A -85,B 0,C 180,E1 19570.539,E2 19570.539} C_VEL
LIN {X 0,Y 411.415,Z 904.404,A -85,B 0,C 180,E1 19574.906,E2 19574.906} C_VEL
LIN {X 0,Y 424.564,Z 862.95,A -85,B 0,C 180,E1 19578.168,E2 19578.168} C_VEL
LIN {X 0,Y 427.629,Z 849.938,A -85,B 0,C 180,E1 19579.05,E2 19579.05} C_VEL
LIN {X 0,Y 419.265,Z 820.247,A -85,B 0,C 180,E1 19583.402,E2 19583.402} C_VEL
LIN {X 0,Y 407.482,Z 791.935,A -85,B 0,C 180,E1 19588.36,E2 19588.36} C_VEL
LIN {X 0,Y 394.986,Z 768.75,A -85,B 0,C 180,E1 19593.573,E2 19593.573} C_VEL
LIN {X 0,Y 383.382,Z 750.731,A -85,B 0,C 180,E1 19599.005,E2 19599.005} C_VEL
LIN {X 0,Y 377.77,Z 743.21,A -85,B 0,C 180,E1 19602.11,E2 19602.11} C_VEL
LIN {X 0,Y 373.933,Z 737.301,A -85,B 0,C 180,E1 19604.723,E2 19604.723} C_VEL
LIN {X 0,Y 369.914,Z 731.048,A -85,B 0,C 180,E1 19608.101,E2 19608.101} C_VEL
LIN {X 0,Y 364.572,Z 722.991,A -85,B 0,C 180,E1 19617.613,E2 19617.613} C_VEL
LIN {X 0,Y 364.819,Z 723.994,A -85,B 0,C 180,E1 19621.632,E2 19621.632} C_VEL
LIN {X 0,Y 368.959,Z 730.12,A -85,B 0,C 180,E1 19628.558,E2 19628.558} C_VEL
LIN {X 0,Y 370.487,Z 732.473,A -85,B 0,C 180,E1 19630.081,E2 19630.081} C_VEL
LIN {X 0,Y 375.733,Z 739.744,A -85,B 0,C 180,E1 19634.093,E2 19634.093} C_VEL
LIN {X 0,Y 382.18,Z 749.104,A -85,B 0,C 180,E1 19637.889,E2 19637.889} C_VEL
LIN {X 0,Y 390.011,Z 760.21,A -85,B 0,C 180,E1 19641.597,E2 19641.597} C_VEL
LIN {X 0,Y 403.02,Z 781.119,A -85,B 0,C 180,E1 19646.892,E2 19646.892} C_VEL
LIN {X 0,Y 416.76,Z 808.995,A -85,B 0,C 180,E1 19652.097,E2 19652.097} C_VEL
LIN {X 0,Y 428.029,Z 840.33,A -85,B 0,C 180,E1 19656.741,E2 19656.741} C_VEL
LIN {X 0,Y 430.238,Z 851.29,A -85,B 0,C 180,E1 19658.074,E2 19658.074} C_VEL
LIN {X 0,Y 418.251,Z 893.458,A -85,B 0,C 180,E1 19660.645,E2 19660.645} C_VEL
LIN {X 0,Y 404.293,Z 934.27,A -85,B 0,C 180,E1 19664.241,E2 19664.241} C_VEL
LIN {X 0,Y 389.298,Z 972.139,A -85,B 0,C 180,E1 19668.93,E2 19668.93} C_VEL
LIN {X 0,Y 375.486,Z 1004.725,A -85,B 0,C 180,E1 19674.584,E2 19674.584} C_VEL
LIN {X 0,Y 364.348,Z 1031.73,A -85,B 0,C 180,E1 19681.159,E2 19681.159} C_VEL
LIN {X 0,Y 356.443,Z 1053.19,A -85,B 0,C 180,E1 19688.627,E2 19688.627} C_VEL
LIN {X 0,Y 352.686,Z 1067.723,A -85,B 0,C 180,E1 19696.329,E2 19696.329} C_VEL
LIN {X 0,Y 351.691,Z 1074.742,A -85,B 0,C 180,E1 19702.572,E2 19702.572} C_VEL
LIN {X 0,Y 351.652,Z 1077.859,A -85,B 0,C 180,E1 19709.999,E2 19709.999} C_VEL
LIN {X 0,Y 351.459,Z 1076.696,A -85,B 0,C 180,E1 19714.946,E2 19714.946} C_VEL
LIN {X 0,Y 352.048,Z 1071.791,A -85,B 0,C 180,E1 19721.168,E2 19721.168} C_VEL
LIN {X 0,Y 354.819,Z 1060.344,A -85,B 0,C 180,E1 19728.681,E2 19728.681} C_VEL
LIN {X 0,Y 360.931,Z 1042.921,A -85,B 0,C 180,E1 19736,E2 19736} C_VEL
LIN {X 0,Y 370.29,Z 1020.8,A -85,B 0,C 180,E1 19742.512,E2 19742.512} C_VEL
LIN {X 0,Y 383.332,Z 992.319,A -85,B 0,C 180,E1 19748.515,E2 19748.515} C_VEL
LIN {X 0,Y 398.444,Z 957.818,A -85,B 0,C 180,E1 19753.735,E2 19753.735} C_VEL
LIN {X 0,Y 413.774,Z 919.373,A -85,B 0,C 180,E1 19757.869,E2 19757.869} C_VEL
LIN {X 0,Y 428.543,Z 875.26,A -85,B 0,C 180,E1 19761.184,E2 19761.184} C_VEL
LIN {X 0,Y 434.841,Z 851.983,A -85,B 0,C 180,E1 19762.503,E2 19762.503} C_VEL
LIN {X 0,Y 429.034,Z 832.724,A -85,B 0,C 180,E1 19765.353,E2 19765.353} C_VEL
LIN {X 0,Y 424.771,Z 826.423,A -85,B 0,C 180,E1 19766.788,E2 19766.788} C_VEL
LIN {X 0,Y 416.708,Z 817.718,A -85,B 0,C 180,E1 19769.335,E2 19769.335} C_VEL
LIN {X 0,Y 405.463,Z 793.867,A -85,B 0,C 180,E1 19774.461,E2 19774.461} C_VEL
LIN {X 0,Y 393.833,Z 773.327,A -85,B 0,C 180,E1 19780.403,E2 19780.403} C_VEL
LIN {X 0,Y 384.986,Z 759.85,A -85,B 0,C 180,E1 19786.344,E2 19786.344} C_VEL
LIN {X 0,Y 380.905,Z 753.276,A -85,B 0,C 180,E1 19790.27,E2 19790.27} C_VEL
LIN {X 0,Y 377.283,Z 746.429,A -85,B 0,C 180,E1 19798.853,E2 19798.853} C_VEL
LIN {X 0,Y 377.409,Z 748.657,A -85,B 0,C 180,E1 19802.018,E2 19802.018} C_VEL
LIN {X 0,Y 381.797,Z 754.78,A -85,B 0,C 180,E1 19809.139,E2 19809.139} C_VEL
LIN {X 0,Y 386.574,Z 762.851,A -85,B 0,C 180,E1 19813.535,E2 19813.535} C_VEL
LIN {X 0,Y 393.727,Z 773.999,A -85,B 0,C 180,E1 19818.227,E2 19818.227} C_VEL
LIN {X 0,Y 404.386,Z 793.834,A -85,B 0,C 180,E1 19824.028,E2 19824.028} C_VEL
LIN {X 0,Y 414.543,Z 816.563,A -85,B 0,C 180,E1 19829.035,E2 19829.035} C_VEL
LIN {X 0,Y 423.476,Z 844.091,A -85,B 0,C 180,E1 19833.913,E2 19833.913} C_VEL
LIN {X 0,Y 426.139,Z 857.703,A -85,B 0,C 180,E1 19835.958,E2 19835.958} C_VEL
LIN {X 0,Y 412.542,Z 898.371,A -85,B 0,C 180,E1 19838.936,E2 19838.936} C_VEL
LIN {X 0,Y 397.572,Z 935.813,A -85,B 0,C 180,E1 19842.801,E2 19842.801} C_VEL
LIN {X 0,Y 382.377,Z 969.471,A -85,B 0,C 180,E1 19847.646,E2 19847.646} C_VEL
LIN {X 0,Y 368.058,Z 998.896,A -85,B 0,C 180,E1 19853.554,E2 19853.554} C_VEL
LIN {X 0,Y 356.567,Z 1022.928,A -85,B 0,C 180,E1 19860.416,E2 19860.416} C_VEL
LIN {X 0,Y 348.604,Z 1041.646,A -85,B 0,C 180,E1 19868.317,E2 19868.317} C_VEL
LIN {X 0,Y 344.844,Z 1053.174,A -85,B 0,C 180,E1 19876.137,E2 19876.137} C_VEL
LIN {X 0,Y 343.588,Z 1058.048,A -85,B 0,C 180,E1 19882.398,E2 19882.398} C_VEL
LIN {X 0,Y 343.785,Z 1059.019,A -85,B 0,C 180,E1 19890.001,E2 19890.001} C_VEL
LIN {X 0,Y 344.252,Z 1054.524,A -85,B 0,C 180,E1 19897.59,E2 19897.59} C_VEL
LIN {X 0,Y 346.602,Z 1045.565,A -85,B 0,C 180,E1 19904.562,E2 19904.562} C_VEL
LIN {X 0,Y 352.214,Z 1029.952,A -85,B 0,C 180,E1 19912.069,E2 19912.069} C_VEL
LIN {X 0,Y 362.088,Z 1007.073,A -85,B 0,C 180,E1 19919.457,E2 19919.457} C_VEL
LIN {X 0,Y 375.081,Z 978.687,A -85,B 0,C 180,E1 19925.828,E2 19925.828} C_VEL
LIN {X 0,Y 390.312,Z 944.174,A -85,B 0,C 180,E1 19931.303,E2 19931.303} C_VEL
LIN {X 0,Y 405.266,Z 906.283,A -85,B 0,C 180,E1 19935.56,E2 19935.56} C_VEL
LIN {X 0,Y 418.809,Z 865.123,A -85,B 0,C 180,E1 19938.858,E2 19938.858} C_VEL
LIN {X 0,Y 421.797,Z 852.989,A -85,B 0,C 180,E1 19939.703,E2 19939.703} C_VEL
LIN {X 0,Y 413.883,Z 823.881,A -85,B 0,C 180,E1 19944.134,E2 19944.134} C_VEL
LIN {X 0,Y 402.791,Z 796.237,A -85,B 0,C 180,E1 19949.169,E2 19949.169} C_VEL
LIN {X 0,Y 391.037,Z 773.967,A -85,B 0,C 180,E1 19954.411,E2 19954.411} C_VEL
LIN {X 0,Y 381.012,Z 757.742,A -85,B 0,C 180,E1 19959.478,E2 19959.478} C_VEL
LIN {X 0,Y 375.613,Z 750.104,A -85,B 0,C 180,E1 19962.686,E2 19962.686} C_VEL
LIN {X 0,Y 372.237,Z 744.776,A -85,B 0,C 180,E1 19965.105,E2 19965.105} C_VEL
LIN {X 0,Y 367.682,Z 737.897,A -85,B 0,C 180,E1 19969.307,E2 19969.307} C_VEL
LIN {X 0,Y 363.592,Z 730.98,A -85,B 0,C 180,E1 19977.607,E2 19977.607} C_VEL
LIN {X 0,Y 363.815,Z 731.799,A -85,B 0,C 180,E1 19981.487,E2 19981.487} C_VEL
LIN {X 0,Y 368.003,Z 737.985,A -85,B 0,C 180,E1 19988.58,E2 19988.58} C_VEL
LIN {X 0,Y 374.188,Z 747.38,A -85,B 0,C 180,E1 19993.817,E2 19993.817} C_VEL
LIN {X 0,Y 383.052,Z 760.096,A -85,B 0,C 180,E1 19998.97,E2 19998.97} C_VEL
LIN {X 0,Y 395.599,Z 780.437,A -85,B 0,C 180,E1 20004.765,E2 20004.765} C_VEL
LIN {X 0,Y 408.02,Z 804.726,A -85,B 0,C 180,E1 20009.862,E2 20009.862} C_VEL
LIN {X 0,Y 418.999,Z 832.506,A -85,B 0,C 180,E1 20014.444,E2 20014.444} C_VEL
LIN {X 0,Y 424.594,Z 853.705,A -85,B 0,C 180,E1 20017.377,E2 20017.377} C_VEL
LIN {X 0,Y 412.165,Z 895.686,A -85,B 0,C 180,E1 20020,E2 20020} C_VEL
LIN {X 0,Y 398.303,Z 934.859,A -85,B 0,C 180,E1 20023.512,E2 20023.512} C_VEL
LIN {X 0,Y 383.407,Z 971.351,A -85,B 0,C 180,E1 20028.062,E2 20028.062} C_VEL
LIN {X 0,Y 368.682,Z 1004.723,A -85,B 0,C 180,E1 20033.912,E2 20033.912} C_VEL
LIN {X 0,Y 357.008,Z 1031.86,A -85,B 0,C 180,E1 20040.65,E2 20040.65} C_VEL
LIN {X 0,Y 348.722,Z 1053.331,A -85,B 0,C 180,E1 20048.322,E2 20048.322} C_VEL
LIN {X 0,Y 344.866,Z 1067.62,A -85,B 0,C 180,E1 20056.107,E2 20056.107} C_VEL
LIN {X 0,Y 343.814,Z 1074.517,A -85,B 0,C 180,E1 20062.4,E2 20062.4} C_VEL
LIN {X 0,Y 343.779,Z 1077.646,A -85,B 0,C 180,E1 20069.999,E2 20069.999} C_VEL
LIN {X 0,Y 343.568,Z 1076.493,A -85,B 0,C 180,E1 20075.06,E2 20075.06} C_VEL
LIN {X 0,Y 344.213,Z 1071.597,A -85,B 0,C 180,E1 20081.425,E2 20081.425} C_VEL
LIN {X 0,Y 347.143,Z 1060.165,A -85,B 0,C 180,E1 20089.11,E2 20089.11} C_VEL
LIN {X 0,Y 353.069,Z 1044.11,A -85,B 0,C 180,E1 20096.099,E2 20096.099} C_VEL
LIN {X 0,Y 362.837,Z 1021.961,A -85,B 0,C 180,E1 20102.883,E2 20102.883} C_VEL
LIN {X 0,Y 376.968,Z 992.246,A -85,B 0,C 180,E1 20109.281,E2 20109.281} C_VEL
LIN {X 0,Y 392.647,Z 957.744,A -85,B 0,C 180,E1 20114.55,E2 20114.55} C_VEL
LIN {X 0,Y 408.43,Z 919.341,A -85,B 0,C 180,E1 20118.705,E2 20118.705} C_VEL
LIN {X 0,Y 423.282,Z 876.321,A -85,B 0,C 180,E1 20121.963,E2 20121.963} C_VEL
LIN {X 0,Y 429.306,Z 855.567,A -85,B 0,C 180,E1 20123.13,E2 20123.13} C_VEL
LIN {X 0,Y 420.557,Z 827.412,A -85,B 0,C 180,E1 20127.594,E2 20127.594} C_VEL
LIN {X 0,Y 416.708,Z 817.718,A -85,B 0,C 180,E1 20129.335,E2 20129.335} C_VEL
LIN {X 0,Y 410.679,Z 811.312,A -85,B 0,C 180,E1 20131.435,E2 20131.435} C_VEL
LIN {X 0,Y 404.625,Z 805.509,A -85,B 0,C 180,E1 20133.627,E2 20133.627} C_VEL
LIN {X 0,Y 394.154,Z 785.511,A -85,B 0,C 180,E1 20139.096,E2 20139.096} C_VEL
LIN {X 0,Y 386.09,Z 772.477,A -85,B 0,C 180,E1 20144.203,E2 20144.203} C_VEL
LIN {X 0,Y 382.818,Z 767.032,A -85,B 0,C 180,E1 20146.848,E2 20146.848} C_VEL
LIN {X 0,Y 379.427,Z 760.965,A -85,B 0,C 180,E1 20150.522,E2 20150.522} C_VEL
LIN {X 0,Y 376.143,Z 754.245,A -85,B 0,C 180,E1 20158.85,E2 20158.85} C_VEL
LIN {X 0,Y 376.465,Z 757.246,A -85,B 0,C 180,E1 20162.888,E2 20162.888} C_VEL
LIN {X 0,Y 380.128,Z 762.548,A -85,B 0,C 180,E1 20168.963,E2 20168.963} C_VEL
LIN {X 0,Y 384.781,Z 770.563,A -85,B 0,C 180,E1 20173.382,E2 20173.382} C_VEL
LIN {X 0,Y 391.27,Z 781.432,A -85,B 0,C 180,E1 20177.981,E2 20177.981} C_VEL
LIN {X 0,Y 401.386,Z 801.082,A -85,B 0,C 180,E1 20183.809,E2 20183.809} C_VEL
LIN {X 0,Y 410.883,Z 824.125,A -85,B 0,C 180,E1 20188.956,E2 20188.956} C_VEL
LIN {X 0,Y 418.86,Z 850.959,A -85,B 0,C 180,E1 20193.769,E2 20193.769} C_VEL
LIN {X 0,Y 420.421,Z 861.322,A -85,B 0,C 180,E1 20195.306,E2 20195.306} C_VEL
LIN {X 0,Y 405.499,Z 903.816,A -85,B 0,C 180,E1 20198.537,E2 20198.537} C_VEL
LIN {X 0,Y 389.408,Z 941.943,A -85,B 0,C 180,E1 20202.693,E2 20202.693} C_VEL
LIN {X 0,Y 374.011,Z 974.341,A -85,B 0,C 180,E1 20207.656,E2 20207.656} C_VEL
LIN {X 0,Y 359.885,Z 1002.105,A -85,B 0,C 180,E1 20213.563,E2 20213.563} C_VEL
LIN {X 0,Y 348.595,Z 1024.823,A -85,B 0,C 180,E1 20220.401,E2 20220.401} C_VEL
LIN {X 0,Y 341.042,Z 1041.815,A -85,B 0,C 180,E1 20227.81,E2 20227.81} C_VEL
LIN {X 0,Y 337.01,Z 1053.5,A -85,B 0,C 180,E1 20235.934,E2 20235.934} C_VEL
LIN {X 0,Y 335.706,Z 1058.249,A -85,B 0,C 180,E1 20242.218,E2 20242.218} C_VEL
LIN {X 0,Y 335.882,Z 1059.234,A -85,B 0,C 180,E1 20250.001,E2 20250.001} C_VEL
LIN {X 0,Y 336.404,Z 1054.76,A -85,B 0,C 180,E1 20257.768,E2 20257.768} C_VEL
LIN {X 0,Y 338.889,Z 1045.825,A -85,B 0,C 180,E1 20264.9,E2 20264.9} C_VEL
LIN {X 0,Y 344.848,Z 1030.051,A -85,B 0,C 180,E1 20272.648,E2 20272.648} C_VEL
LIN {X 0,Y 355.105,Z 1007.379,A -85,B 0,C 180,E1 20280.096,E2 20280.096} C_VEL
LIN {X 0,Y 368.468,Z 979.325,A -85,B 0,C 180,E1 20286.497,E2 20286.497} C_VEL
LIN {X 0,Y 383.714,Z 945.932,A -85,B 0,C 180,E1 20291.896,E2 20291.896} C_VEL
LIN {X 0,Y 398.51,Z 909.823,A -85,B 0,C 180,E1 20296.067,E2 20296.067} C_VEL
LIN {X 0,Y 411.885,Z 871.184,A -85,B 0,C 180,E1 20299.301,E2 20299.301} C_VEL
LIN {X 0,Y 416.073,Z 856.535,A -85,B 0,C 180,E1 20300.31,E2 20300.31} C_VEL
LIN {X 0,Y 408.549,Z 827.421,A -85,B 0,C 180,E1 20304.9,E2 20304.9} C_VEL
LIN {X 0,Y 397.812,Z 799.851,A -85,B 0,C 180,E1 20310.155,E2 20310.155} C_VEL
LIN {X 0,Y 386.344,Z 777.503,A -85,B 0,C 180,E1 20315.687,E2 20315.687} C_VEL
LIN {X 0,Y 377.013,Z 762.416,A -85,B 0,C 180,E1 20320.858,E2 20320.858} C_VEL
LIN {X 0,Y 370.527,Z 752.208,A -85,B 0,C 180,E1 20325.489,E2 20325.489} C_VEL
LIN {X 0,Y 366.313,Z 745.584,A -85,B 0,C 180,E1 20329.568,E2 20329.568} C_VEL
LIN {X 0,Y 362.567,Z 738.703,A -85,B 0,C 180,E1 20338.798,E2 20338.798} C_VEL
LIN {X 0,Y 362.843,Z 740.09,A -85,B 0,C 180,E1 20341.641,E2 20341.641} C_VEL
LIN {X 0,Y 367.619,Z 747.238,A -85,B 0,C 180,E1 20349.337,E2 20349.337} C_VEL
LIN {X 0,Y 372.73,Z 755.287,A -85,B 0,C 180,E1 20353.665,E2 20353.665} C_VEL
LIN {X 0,Y 380.798,Z 767.36,A -85,B 0,C 180,E1 20358.635,E2 20358.635} C_VEL
LIN {X 0,Y 392.937,Z 787.888,A -85,B 0,C 180,E1 20364.564,E2 20364.564} C_VEL
LIN {X 0,Y 405.238,Z 813.398,A -85,B 0,C 180,E1 20369.909,E2 20369.909} C_VEL
LIN {X 0,Y 415.604,Z 842.661,A -85,B 0,C 180,E1 20374.726,E2 20374.726} C_VEL
LIN {X 0,Y 418.823,Z 856.812,A -85,B 0,C 180,E1 20376.695,E2 20376.695} C_VEL
LIN {X 0,Y 405.879,Z 898.653,A -85,B 0,C 180,E1 20379.393,E2 20379.393} C_VEL
LIN {X 0,Y 391.785,Z 936.793,A -85,B 0,C 180,E1 20382.903,E2 20382.903} C_VEL
LIN {X 0,Y 376.921,Z 972.026,A -85,B 0,C 180,E1 20387.393,E2 20387.393} C_VEL
LIN {X 0,Y 362.23,Z 1004.125,A -85,B 0,C 180,E1 20393.085,E2 20393.085} C_VEL
LIN {X 0,Y 349.835,Z 1031.688,A -85,B 0,C 180,E1 20400.027,E2 20400.027} C_VEL
LIN {X 0,Y 341.17,Z 1053.069,A -85,B 0,C 180,E1 20407.817,E2 20407.817} C_VEL
LIN {X 0,Y 337.034,Z 1067.548,A -85,B 0,C 180,E1 20415.895,E2 20415.895} C_VEL
LIN {X 0,Y 335.792,Z 1074.883,A -85,B 0,C 180,E1 20423.095,E2 20423.095} C_VEL
LIN {X 0,Y 335.878,Z 1077.432,A -85,B 0,C 180,E1 20429.999,E2 20429.999} C_VEL
LIN {X 0,Y 335.74,Z 1075.427,A -85,B 0,C 180,E1 20436.832,E2 20436.832} C_VEL
LIN {X 0,Y 337.029,Z 1068.517,A -85,B 0,C 180,E1 20444.107,E2 20444.107} C_VEL
LIN {X 0,Y 340.873,Z 1056.164,A -85,B 0,C 180,E1 20451.515,E2 20451.515} C_VEL
LIN {X 0,Y 348.705,Z 1037.427,A -85,B 0,C 180,E1 20458.986,E2 20458.986} C_VEL
LIN {X 0,Y 360.128,Z 1013.668,A -85,B 0,C 180,E1 20465.618,E2 20465.618} C_VEL
LIN {X 0,Y 375.498,Z 982.087,A -85,B 0,C 180,E1 20471.839,E2 20471.839} C_VEL
LIN {X 0,Y 392.193,Z 945.894,A -85,B 0,C 180,E1 20476.827,E2 20476.827} C_VEL
LIN {X 0,Y 408.602,Z 905.072,A -85,B 0,C 180,E1 20480.778,E2 20480.778} C_VEL
LIN {X 0,Y 423.129,Z 860.836,A -85,B 0,C 180,E1 20483.727,E2 20483.727} C_VEL
LIN {X 0,Y 422.901,Z 855.61,A -85,B 0,C 180,E1 20484.31,E2 20484.31} C_VEL
LIN {X 0,Y 414.302,Z 828.014,A -85,B 0,C 180,E1 20488.952,E2 20488.952} C_VEL
LIN {X 0,Y 404.625,Z 805.509,A -85,B 0,C 180,E1 20493.627,E2 20493.627} C_VEL
LIN {X 0,Y 398.876,Z 800.661,A -85,B 0,C 180,E1 20495.884,E2 20495.884} C_VEL
LIN {X 0,Y 393.435,Z 796.515,A -85,B 0,C 180,E1 20498.246,E2 20498.246} C_VEL
LIN {X 0,Y 385.33,Z 781.58,A -85,B 0,C 180,E1 20503.514,E2 20503.514} C_VEL
LIN {X 0,Y 380.513,Z 774.015,A -85,B 0,C 180,E1 20507.498,E2 20507.498} C_VEL
LIN {X 0,Y 377.697,Z 768.576,A -85,B 0,C 180,E1 20510.769,E2 20510.769} C_VEL
LIN {X 0,Y 374.805,Z 762.03,A -85,B 0,C 180,E1 20518.846,E2 20518.846} C_VEL
LIN {X 0,Y 378.425,Z 770.25,A -85,B 0,C 180,E1 20528.786,E2 20528.786} C_VEL
LIN {X 0,Y 382.862,Z 778.517,A -85,B 0,C 180,E1 20533.378,E2 20533.378} C_VEL
LIN {X 0,Y 388.85,Z 789.036,A -85,B 0,C 180,E1 20537.803,E2 20537.803} C_VEL
LIN {X 0,Y 397.746,Z 807.456,A -85,B 0,C 180,E1 20543.377,E2 20543.377} C_VEL
LIN {X 0,Y 406.789,Z 830.691,A -85,B 0,C 180,E1 20548.665,E2 20548.665} C_VEL
LIN {X 0,Y 413.917,Z 857.065,A -85,B 0,C 180,E1 20553.508,E2 20553.508} C_VEL
LIN {X 0,Y 415.043,Z 863.79,A -85,B 0,C 180,E1 20554.57,E2 20554.57} C_VEL
LIN {X 0,Y 399.497,Z 906.365,A -85,B 0,C 180,E1 20557.865,E2 20557.865} C_VEL
LIN {X 0,Y 382.657,Z 944.859,A -85,B 0,C 180,E1 20562.176,E2 20562.176} C_VEL
LIN {X 0,Y 365.646,Z 979.139,A -85,B 0,C 180,E1 20567.666,E2 20567.666} C_VEL
LIN {X 0,Y 350.455,Z 1007.92,A -85,B 0,C 180,E1 20574.287,E2 20574.287} C_VEL
LIN {X 0,Y 339.418,Z 1029.184,A -85,B 0,C 180,E1 20581.319,E2 20581.319} C_VEL
LIN {X 0,Y 332.315,Z 1045.025,A -85,B 0,C 180,E1 20589.091,E2 20589.091} C_VEL
LIN {X 0,Y 328.872,Z 1054.68,A -85,B 0,C 180,E1 20596.681,E2 20596.681} C_VEL
LIN {X 0,Y 327.628,Z 1059.425,A -85,B 0,C 180,E1 20604.693,E2 20604.693} C_VEL
LIN {X 0,Y 328.008,Z 1059.447,A -85,B 0,C 180,E1 20610.001,E2 20610.001} C_VEL
LIN {X 0,Y 328.534,Z 1054.998,A -85,B 0,C 180,E1 20617.955,E2 20617.955} C_VEL
LIN {X 0,Y 331.172,Z 1046.087,A -85,B 0,C 180,E1 20625.256,E2 20625.256} C_VEL
LIN {X 0,Y 337.473,Z 1030.329,A -85,B 0,C 180,E1 20633.171,E2 20633.171} C_VEL
LIN {X 0,Y 348.171,Z 1007.683,A -85,B 0,C 180,E1 20640.759,E2 20640.759} C_VEL
